      GB2 : Array[0..7480] of Word := [16#A1E8, 16#A1EC, 16#A1A7, 16#A1E3, 16#A1C0, 16#A1A4, 16#A1C1, 16#A8A4, 16#A8A2, 16#A8A8, 16#A8A6, 16#A8BA, 16#A8AC, 16#A8AA, 16#A8B0, 16#A8AE, 16#A1C2, 16#A8B4, 16#A8B2, 16#A8B9, 16#A8A1, 16#A8A5, 16#A8A7, 16#A8A9, 16#A8BD, 16#A8BE, 16#A8AD, 16#A8B1, 16#A8A3, 16#A8AB, 16#A8AF, 16#A8B3, 16#A8B5, 16#A8B6, 16#A8B7, 16#A8B8, 16#A8BB, 16#A8C0, 16#A1A6, 16#A1A5, 16#A6A1, 16#A6A2, 16#A6A3, 16#A6A4, 16#A6A5, 16#A6A6, 16#A6A7, 16#A6A8, 16#A6A9, 16#A6AA, 16#A6AB, 16#A6AC, 16#A6AD, 16#A6AE, 16#A6AF, 16#A6B0, 16#A6B1, 16#A6B2, 16#A6B3, 16#A6B4, 16#A6B5, 16#A6B6, 16#A6B7, 16#A6B8, 16#A6C1, 16#A6C2, 16#A6C3, 16#A6C4, 16#A6C5, 16#A6C6, 16#A6C7, 16#A6C8, 16#A6C9, 16#A6CA, 16#A6CB, 16#A6CC, 16#A6CD, 16#A6CE, 16#A6CF, 16#A6D0, 16#A6D1, 16#A6D2, 16#A6D3, 16#A6D4, 16#A6D5, 16#A6D6, 16#A6D7, 16#A6D8, 16#A7A7, 16#A7A1, 16#A7A2, 16#A7A3, 16#A7A4, 16#A7A5, 16#A7A6, 16#A7A8, 16#A7A9, 16#A7AA, 16#A7AB, 16#A7AC, 16#A7AD, 16#A7AE, 16#A7AF, 16#A7B0, 16#A7B1, 16#A7B2, 16#A7B3, 16#A7B4, 16#A7B5, 16#A7B6, 16#A7B7, 16#A7B8, 16#A7B9, 16#A7BA, 16#A7BB, 16#A7BC, 16#A7BD, 16#A7BE, 16#A7BF, 16#A7C0, 16#A7C1, 16#A7D1, 16#A7D2, 16#A7D3, 16#A7D4, 16#A7D5, 16#A7D6, 16#A7D8, 16#A7D9, 16#A7DA, 16#A7DB, 16#A7DC, 16#A7DD, 16#A7DE, 16#A7DF, 16#A7E0, 16#A7E1, 16#A7E2, 16#A7E3, 16#A7E4, 16#A7E5, 16#A7E6, 16#A7E7, 16#A7E8, 16#A7E9, 16#A7EA, 16#A7EB, 16#A7EC, 16#A7ED, 16#A7EE, 16#A7EF, 16#A7F0, 16#A7F1, 16#A7D7, 16#A1AA, 16#A1AC, 16#A1AE, 16#A1AF, 16#A1B0, 16#A1B1, 16#A1AD, 16#A1EB, 16#A1E4, 16#A1E5, 16#A1F9, 16#A1E6, 16#A1ED, 16#A2F1, 16#A2F2, 16#A2F3, 16#A2F4, 16#A2F5, 16#A2F6, 16#A2F7, 16#A2F8, 16#A2F9, 16#A2FA, 16#A2FB, 16#A2FC, 16#A2A1, 16#A2A2, 16#A2A3, 16#A2A4, 16#A2A5, 16#A2A6, 16#A2A7, 16#A2A8, 16#A2A9, 16#A2AA, 16#A1FB, 16#A1FC, 16#A1FA, 16#A1FD, 16#A1CA, 16#A1C7, 16#A1C6, 16#A1CC, 16#A1D8, 16#A1DE, 16#A1CF, 16#A1CE, 16#A1C4, 16#A1C5, 16#A1C9, 16#A1C8, 16#A1D2, 16#A1D3, 16#A1E0, 16#A1DF, 16#A1C3, 16#A1CB, 16#A1D7, 16#A1D6, 16#A1D5, 16#A1D9, 16#A1D4, 16#A1DC, 16#A1DD, 16#A1DA, 16#A1DB, 16#A1D1, 16#A1CD, 16#A1D0, 16#A2D9, 16#A2DA, 16#A2DB, 16#A2DC, 16#A2DD, 16#A2DE, 16#A2DF, 16#A2E0, 16#A2E1, 16#A2E2, 16#A2C5, 16#A2C6, 16#A2C7, 16#A2C8, 16#A2C9, 16#A2CA, 16#A2CB, 16#A2CC, 16#A2CD, 16#A2CE, 16#A2CF, 16#A2D0, 16#A2D1, 16#A2D2, 16#A2D3, 16#A2D4, 16#A2D5, 16#A2D6, 16#A2D7, 16#A2D8, 16#A2B1, 16#A2B2, 16#A2B3, 16#A2B4, 16#A2B5, 16#A2B6, 16#A2B7, 16#A2B8, 16#A2B9, 16#A2BA, 16#A2BB, 16#A2BC, 16#A2BD, 16#A2BE, 16#A2BF, 16#A2C0, 16#A2C1, 16#A2C2, 16#A2C3, 16#A2C4, 16#A9A4, 16#A9A5, 16#A9A6, 16#A9A7, 16#A9A8, 16#A9A9, 16#A9AA, 16#A9AB, 16#A9AC, 16#A9AD, 16#A9AE, 16#A9AF, 16#A9B0, 16#A9B1, 16#A9B2, 16#A9B3, 16#A9B4, 16#A9B5, 16#A9B6, 16#A9B7, 16#A9B8, 16#A9B9, 16#A9BA, 16#A9BB, 16#A9BC, 16#A9BD, 16#A9BE, 16#A9BF, 16#A9C0, 16#A9C1, 16#A9C2, 16#A9C3, 16#A9C4, 16#A9C5, 16#A9C6, 16#A9C7, 16#A9C8, 16#A9C9, 16#A9CA, 16#A9CB, 16#A9CC, 16#A9CD, 16#A9CE, 16#A9CF, 16#A9D0, 16#A9D1, 16#A9D2, 16#A9D3, 16#A9D4, 16#A9D5, 16#A9D6, 16#A9D7, 16#A9D8, 16#A9D9, 16#A9DA, 16#A9DB, 16#A9DC, 16#A9DD, 16#A9DE, 16#A9DF, 16#A9E0, 16#A9E1, 16#A9E2, 16#A9E3, 16#A9E4, 16#A9E5, 16#A9E6, 16#A9E7, 16#A9E8, 16#A9E9, 16#A9EA, 16#A9EB, 16#A9EC, 16#A9ED, 16#A9EE, 16#A9EF, 16#A1F6, 16#A1F5, 16#A1F8, 16#A1F7, 16#A1F4, 16#A1F3, 16#A1F0, 16#A1F2, 16#A1F1, 16#A1EF, 16#A1EE, 16#A1E2, 16#A1E1, 16#A1A1, 16#A1A2, 16#A1A3, 16#A1A8, 16#A1A9, 16#A1B4, 16#A1B5, 16#A1B6, 16#A1B7, 16#A1B8, 16#A1B9, 16#A1BA, 16#A1BB, 16#A1BE, 16#A1BF, 16#A1FE, 16#A1B2, 16#A1B3, 16#A1BC, 16#A1BD, 16#A4A1, 16#A4A2, 16#A4A3, 16#A4A4, 16#A4A5, 16#A4A6, 16#A4A7, 16#A4A8, 16#A4A9, 16#A4AA, 16#A4AB, 16#A4AC, 16#A4AD, 16#A4AE, 16#A4AF, 16#A4B0, 16#A4B1, 16#A4B2, 16#A4B3, 16#A4B4, 16#A4B5, 16#A4B6, 16#A4B7, 16#A4B8, 16#A4B9, 16#A4BA, 16#A4BB, 16#A4BC, 16#A4BD, 16#A4BE, 16#A4BF, 16#A4C0, 16#A4C1, 16#A4C2, 16#A4C3, 16#A4C4, 16#A4C5, 16#A4C6, 16#A4C7, 16#A4C8, 16#A4C9, 16#A4CA, 16#A4CB, 16#A4CC, 16#A4CD, 16#A4CE, 16#A4CF, 16#A4D0, 16#A4D1, 16#A4D2, 16#A4D3, 16#A4D4, 16#A4D5, 16#A4D6, 16#A4D7, 16#A4D8, 16#A4D9, 16#A4DA, 16#A4DB, 16#A4DC, 16#A4DD, 16#A4DE, 16#A4DF, 16#A4E0, 16#A4E1, 16#A4E2, 16#A4E3, 16#A4E4, 16#A4E5, 16#A4E6, 16#A4E7, 16#A4E8, 16#A4E9, 16#A4EA, 16#A4EB, 16#A4EC, 16#A4ED, 16#A4EE, 16#A4EF, 16#A4F0, 16#A4F1, 16#A4F2, 16#A4F3, 16#A5A1, 16#A5A2, 16#A5A3, 16#A5A4, 16#A5A5, 16#A5A6, 16#A5A7, 16#A5A8, 16#A5A9, 16#A5AA, 16#A5AB, 16#A5AC, 16#A5AD, 16#A5AE, 16#A5AF, 16#A5B0, 16#A5B1, 16#A5B2, 16#A5B3, 16#A5B4, 16#A5B5, 16#A5B6, 16#A5B7, 16#A5B8, 16#A5B9, 16#A5BA, 16#A5BB, 16#A5BC, 16#A5BD, 16#A5BE, 16#A5BF, 16#A5C0, 16#A5C1, 16#A5C2, 16#A5C3, 16#A5C4, 16#A5C5, 16#A5C6, 16#A5C7, 16#A5C8, 16#A5C9, 16#A5CA, 16#A5CB, 16#A5CC, 16#A5CD, 16#A5CE, 16#A5CF, 16#A5D0, 16#A5D1, 16#A5D2, 16#A5D3, 16#A5D4, 16#A5D5, 16#A5D6, 16#A5D7, 16#A5D8, 16#A5D9, 16#A5DA, 16#A5DB, 16#A5DC, 16#A5DD, 16#A5DE, 16#A5DF, 16#A5E0, 16#A5E1, 16#A5E2, 16#A5E3, 16#A5E4, 16#A5E5, 16#A5E6, 16#A5E7, 16#A5E8, 16#A5E9, 16#A5EA, 16#A5EB, 16#A5EC, 16#A5ED, 16#A5EE, 16#A5EF, 16#A5F0, 16#A5F1, 16#A5F2, 16#A5F3, 16#A5F4, 16#A5F5, 16#A5F6, 16#A8C5, 16#A8C6, 16#A8C7, 16#A8C8, 16#A8C9, 16#A8CA, 16#A8CB, 16#A8CC, 16#A8CD, 16#A8CE, 16#A8CF, 16#A8D0, 16#A8D1, 16#A8D2, 16#A8D3, 16#A8D4, 16#A8D5, 16#A8D6, 16#A8D7, 16#A8D8, 16#A8D9, 16#A8DA, 16#A8DB, 16#A8DC, 16#A8DD, 16#A8DE, 16#A8DF, 16#A8E0, 16#A8E1, 16#A8E2, 16#A8E3, 16#A8E4, 16#A8E5, 16#A8E6, 16#A8E7, 16#A8E8, 16#A8E9, 16#A2E5, 16#A2E6, 16#A2E7, 16#A2E8, 16#A2E9, 16#A2EA, 16#A2EB, 16#A2EC, 16#A2ED, 16#A2EE, 16#D2BB, 16#B6A1, 16#C6DF, 16#CDF2, 16#D5C9, 16#C8FD, 16#C9CF, 16#CFC2, 16#D8A2, 16#B2BB, 16#D3EB, 16#D8A4, 16#B3F3, 16#D7A8, 16#C7D2, 16#D8A7, 16#CAC0, 16#C7F0, 16#B1FB, 16#D2B5, 16#B4D4, 16#B6AB, 16#CBBF, 16#D8A9, 16#B6AA, 16#C1BD, 16#D1CF, 16#C9A5, 16#D8AD, 16#B8F6, 16#D1BE, 16#E3DC, 16#D6D0, 16#B7E1, 16#B4AE, 16#C1D9, 16#D8BC, 16#CDE8, 16#B5A4, 16#CEAA, 16#D6F7, 16#C0F6, 16#BED9, 16#D8AF, 16#C4CB, 16#BEC3, 16#D8B1, 16#C3B4, 16#D2E5, 16#D6AE, 16#CEDA, 16#D5A7, 16#BAF5, 16#B7A6, 16#C0D6, 16#C6B9, 16#C5D2, 16#C7C7, 16#B9D4, 16#B3CB, 16#D2D2, 16#D8BF, 16#BEC5, 16#C6F2, 16#D2B2, 16#CFB0, 16#CFE7, 16#CAE9, 16#D8C0, 16#C2F2, 16#C2D2, 16#C8E9, 16#C7AC, 16#C1CB, 16#D3E8, 16#D5F9, 16#CAC2, 16#B6FE, 16#D8A1, 16#D3DA, 16#BFF7, 16#D4C6, 16#BBA5, 16#D8C1, 16#CEE5, 16#BEAE, 16#D8A8, 16#D1C7, 16#D0A9, 16#D8BD, 16#D9EF, 16#CDF6, 16#BFBA, 16#BDBB, 16#BAA5, 16#D2E0, 16#B2FA, 16#BAE0, 16#C4B6, 16#CFED, 16#BEA9, 16#CDA4, 16#C1C1, 16#C7D7, 16#D9F1, 16#D9F4, 16#C8CB, 16#D8E9, 16#D2DA, 16#CAB2, 16#C8CA, 16#D8EC, 16#D8EA, 16#D8C6, 16#BDF6, 16#C6CD, 16#B3F0, 16#D8EB, 16#BDF1, 16#BDE9, 16#C8D4, 16#B4D3, 16#C2D8, 16#B2D6, 16#D7D0, 16#CACB, 16#CBFB, 16#D5CC, 16#B8B6, 16#CFC9, 16#D9DA, 16#D8F0, 16#C7AA, 16#D8EE, 16#B4FA, 16#C1EE, 16#D2D4, 16#D8ED, 16#D2C7, 16#D8EF, 16#C3C7, 16#D1F6, 16#D6D9, 16#D8F2, 16#D8F5, 16#BCFE, 16#BCDB, 16#C8CE, 16#B7DD, 16#B7C2, 16#C6F3, 16#D8F8, 16#D2C1, 16#CEE9, 16#BCBF, 16#B7FC, 16#B7A5, 16#D0DD, 16#D6DA, 16#D3C5, 16#BBEF, 16#BBE1, 16#D8F1, 16#C9A1, 16#CEB0, 16#B4AB, 16#D8F3, 16#C9CB, 16#D8F6, 16#C2D7, 16#D8F7, 16#CEB1, 16#D8F9, 16#B2AE, 16#B9C0, 16#D9A3, 16#B0E9, 16#C1E6, 16#C9EC, 16#CBC5, 16#CBC6, 16#D9A4, 16#B5E8, 16#B5AB, 16#CEBB, 16#B5CD, 16#D7A1, 16#D7F4, 16#D3D3, 16#CCE5, 16#BACE, 16#D9A2, 16#D9DC, 16#D3E0, 16#D8FD, 16#B7F0, 16#D7F7, 16#D8FE, 16#D8FA, 16#D9A1, 16#C4E3, 16#D3B6, 16#D8F4, 16#D9DD, 16#D8FB, 16#C5E5, 16#C0D0, 16#D1F0, 16#B0DB, 16#BCD1, 16#D9A6, 16#D9A5, 16#D9AC, 16#D9AE, 16#D9AB, 16#CAB9, 16#D9A9, 16#D6B6, 16#B3DE, 16#D9A8, 16#C0FD, 16#CACC, 16#D9AA, 16#D9A7, 16#D9B0, 16#B6B1, 16#B9A9, 16#D2C0, 16#CFC0, 16#C2C2, 16#BDC4, 16#D5EC, 16#B2E0, 16#C7C8, 16#BFEB, 16#D9AD, 16#D9AF, 16#CEEA, 16#BAEE, 16#C7D6, 16#B1E3, 16#B4D9, 16#B6ED, 16#D9B4, 16#BFA1, 16#D9DE, 16#C7CE, 16#C0FE, 16#D9B8, 16#CBD7, 16#B7FD, 16#D9B5, 16#D9B7, 16#B1A3, 16#D3E1, 16#D9B9, 16#D0C5, 16#D9B6, 16#D9B1, 16#D9B2, 16#C1A9, 16#D9B3, 16#BCF3, 16#D0DE, 16#B8A9, 16#BEE3, 16#D9BD, 16#D9BA, 16#B0B3, 16#D9C2, 16#D9C4, 16#B1B6, 16#D9BF, 16#B5B9, 16#BEF3, 16#CCC8, 16#BAF2, 16#D2D0, 16#D9C3, 16#BDE8, 16#B3AB, 16#D9C5, 16#BEEB, 16#D9C6, 16#D9BB, 16#C4DF, 16#D9BE, 16#D9C1, 16#D9C0, 16#D5AE, 16#D6B5, 16#C7E3, 16#D9C8, 16#BCD9, 16#D9CA, 16#D9BC, 16#D9CB, 16#C6AB, 16#D9C9, 16#D7F6, 16#CDA3, 16#BDA1, 16#D9CC, 16#C5BC, 16#CDB5, 16#D9CD, 16#D9C7, 16#B3A5, 16#BFFE, 16#B8B5, 16#C0FC, 16#B0F8, 16#B4F6, 16#D9CE, 16#D9CF, 16#B4A2, 16#D9D0, 16#B4DF, 16#B0C1, 16#D9D1, 16#C9B5, 16#CFF1, 16#D9D2, 16#C1C5, 16#D9D6, 16#C9AE, 16#D9D5, 16#D9D4, 16#D9D7, 16#CBDB, 16#BDA9, 16#C6A7, 16#D9D3, 16#D9D8, 16#D9D9, 16#C8E5, 16#C0DC, 16#B6F9, 16#D8A3, 16#D4CA, 16#D4AA, 16#D0D6, 16#B3E4, 16#D5D7, 16#CFC8, 16#B9E2, 16#BFCB, 16#C3E2, 16#B6D2, 16#CDC3, 16#D9EE, 16#D9F0, 16#B5B3, 16#B6B5, 16#BEA4, 16#C8EB, 16#C8AB, 16#B0CB, 16#B9AB, 16#C1F9, 16#D9E2, 16#C0BC, 16#B9B2, 16#B9D8, 16#D0CB, 16#B1F8, 16#C6E4, 16#BEDF, 16#B5E4, 16#D7C8, 16#D1F8, 16#BCE6, 16#CADE, 16#BCBD, 16#D9E6, 16#D8E7, 16#C4DA, 16#B8D4, 16#C8BD, 16#B2E1, 16#D4D9, 16#C3B0, 16#C3E1, 16#DAA2, 16#C8DF, 16#D0B4, 16#BEFC, 16#C5A9, 16#B9DA, 16#DAA3, 16#D4A9, 16#DAA4, 16#D9FB, 16#B6AC, 16#B7EB, 16#B1F9, 16#D9FC, 16#B3E5, 16#BEF6, 16#BFF6, 16#D2B1, 16#C0E4, 16#B6B3, 16#D9FE, 16#D9FD, 16#BEBB, 16#C6E0, 16#D7BC, 16#DAA1, 16#C1B9, 16#B5F2, 16#C1E8, 16#BCF5, 16#B4D5, 16#C1DD, 16#C4FD, 16#BCB8, 16#B7B2, 16#B7EF, 16#D9EC, 16#C6BE, 16#BFAD, 16#BBCB, 16#B5CA, 16#DBC9, 16#D0D7, 16#CDB9, 16#B0BC, 16#B3F6, 16#BBF7, 16#DBCA, 16#BAAF, 16#D4E4, 16#B5B6, 16#B5F3, 16#D8D6, 16#C8D0, 16#B7D6, 16#C7D0, 16#D8D7, 16#BFAF, 16#DBBB, 16#D8D8, 16#D0CC, 16#BBAE, 16#EBBE, 16#C1D0, 16#C1F5, 16#D4F2, 16#B8D5, 16#B4B4, 16#B3F5, 16#C9BE, 16#C5D0, 16#C5D9, 16#C0FB, 16#B1F0, 16#D8D9, 16#B9CE, 16#B5BD, 16#D8DA, 16#D6C6, 16#CBA2, 16#C8AF, 16#C9B2, 16#B4CC, 16#BFCC, 16#B9F4, 16#D8DB, 16#D8DC, 16#B6E7, 16#BCC1, 16#CCEA, 16#CFF7, 16#D8DD, 16#C7B0, 16#B9D0, 16#BDA3, 16#CCDE, 16#C6CA, 16#D8E0, 16#D8DE, 16#D8DF, 16#B0FE, 16#BEE7, 16#CAA3, 16#BCF4, 16#B8B1, 16#B8EE, 16#D8E2, 16#BDCB, 16#D8E4, 16#D8E3, 16#C5FC, 16#D8E5, 16#D8E6, 16#C1A6, 16#C8B0, 16#B0EC, 16#B9A6, 16#BCD3, 16#CEF1, 16#DBBD, 16#C1D3, 16#B6AF, 16#D6FA, 16#C5AC, 16#BDD9, 16#DBBE, 16#DBBF, 16#C0F8, 16#BEA2, 16#C0CD, 16#DBC0, 16#CAC6, 16#B2AA, 16#D3C2, 16#C3E3, 16#D1AB, 16#DBC2, 16#C0D5, 16#DBC3, 16#BFB1, 16#C4BC, 16#C7DA, 16#DBC4, 16#D9E8, 16#C9D7, 16#B9B4, 16#CEF0, 16#D4C8, 16#B0FC, 16#B4D2, 16#D0D9, 16#D9E9, 16#DECB, 16#D9EB, 16#D8B0, 16#BBAF, 16#B1B1, 16#B3D7, 16#D8CE, 16#D4D1, 16#BDB3, 16#BFEF, 16#CFBB, 16#D8D0, 16#B7CB, 16#D8D1, 16#C6A5, 16#C7F8, 16#D2BD, 16#D8D2, 16#C4E4, 16#CAAE, 16#C7A7, 16#D8A6, 16#C9FD, 16#CEE7, 16#BBDC, 16#B0EB, 16#BBAA, 16#D0AD, 16#B1B0, 16#D7E4, 16#D7BF, 16#B5A5, 16#C2F4, 16#C4CF, 16#B2A9, 16#B2B7, 16#B1E5, 16#DFB2, 16#D5BC, 16#BFA8, 16#C2AC, 16#D8D5, 16#C2B1, 16#D8D4, 16#CED4, 16#DAE0, 16#CEC0, 16#D8B4, 16#C3AE, 16#D3A1, 16#CEA3, 16#BCB4, 16#C8B4, 16#C2D1, 16#BEED, 16#D0B6, 16#DAE1, 16#C7E4, 16#B3A7, 16#B6F2, 16#CCFC, 16#C0FA, 16#C0F7, 16#D1B9, 16#D1E1, 16#D8C7, 16#B2DE, 16#C0E5, 16#BAF1, 16#D8C8, 16#D4AD, 16#CFE1, 16#D8C9, 16#D8CA, 16#CFC3, 16#B3F8, 16#BEC7, 16#D8CB, 16#DBCC, 16#C8A5, 16#CFD8, 16#C8FE, 16#B2CE, 16#D3D6, 16#B2E6, 16#BCB0, 16#D3D1, 16#CBAB, 16#B7B4, 16#B7A2, 16#CAE5, 16#C8A1, 16#CADC, 16#B1E4, 16#D0F0, 16#C5D1, 16#DBC5, 16#B5FE, 16#BFDA, 16#B9C5, 16#BEE4, 16#C1ED, 16#DFB6, 16#DFB5, 16#D6BB, 16#BDD0, 16#D5D9, 16#B0C8, 16#B6A3, 16#BFC9, 16#CCA8, 16#DFB3, 16#CAB7, 16#D3D2, 16#D8CF, 16#D2B6, 16#BAC5, 16#CBBE, 16#CCBE, 16#DFB7, 16#B5F0, 16#DFB4, 16#D3F5, 16#B3D4, 16#B8F7, 16#DFBA, 16#BACF, 16#BCAA, 16#B5F5, 16#CDAC, 16#C3FB, 16#BAF3, 16#C0F4, 16#CDC2, 16#CFF2, 16#DFB8, 16#CFC5, 16#C2C0, 16#DFB9, 16#C2F0, 16#BEFD, 16#C1DF, 16#CDCC, 16#D2F7, 16#B7CD, 16#DFC1, 16#DFC4, 16#B7F1, 16#B0C9, 16#B6D6, 16#B7D4, 16#BAAC, 16#CCFD, 16#BFD4, 16#CBB1, 16#C6F4, 16#D6A8, 16#DFC5, 16#CEE2, 16#B3B3, 16#CEFC, 16#B4B5, 16#CEC7, 16#BAF0, 16#CEE1, 16#D1BD, 16#DFC0, 16#B4F4, 16#B3CA, 16#B8E6, 16#DFBB, 16#C4C5, 16#DFBC, 16#DFBD, 16#DFBE, 16#C5BB, 16#DFBF, 16#DFC2, 16#D4B1, 16#DFC3, 16#C7BA, 16#CED8, 16#C4D8, 16#DFCA, 16#DFCF, 16#D6DC, 16#DFC9, 16#DFDA, 16#CEB6, 16#BAC7, 16#DFCE, 16#DFC8, 16#C5DE, 16#C9EB, 16#BAF4, 16#C3FC, 16#BED7, 16#DFC6, 16#DFCD, 16#C5D8, 16#D5A6, 16#BACD, 16#BECC, 16#D3BD, 16#B8C0, 16#D6E4, 16#DFC7, 16#B9BE, 16#BFA7, 16#C1FC, 16#DFCB, 16#DFCC, 16#DFD0, 16#DFDB, 16#DFE5, 16#DFD7, 16#DFD6, 16#D7C9, 16#DFE3, 16#DFE4, 16#E5EB, 16#D2A7, 16#DFD2, 16#BFA9, 16#D4DB, 16#BFC8, 16#DFD4, 16#CFCC, 16#DFDD, 16#D1CA, 16#DFDE, 16#B0A7, 16#C6B7, 16#DFD3, 16#BAE5, 16#B6DF, 16#CDDB, 16#B9FE, 16#D4D5, 16#DFDF, 16#CFEC, 16#B0A5, 16#DFE7, 16#DFD1, 16#D1C6, 16#DFD5, 16#DFD8, 16#DFD9, 16#DFDC, 16#BBA9, 16#DFE0, 16#DFE1, 16#DFE2, 16#DFE6, 16#DFE8, 16#D3B4, 16#B8E7, 16#C5B6, 16#DFEA, 16#C9DA, 16#C1A8, 16#C4C4, 16#BFDE, 16#CFF8, 16#D5DC, 16#DFEE, 16#B2B8, 16#BADF, 16#DFEC, 16#DBC1, 16#D1E4, 16#CBF4, 16#B4BD, 16#B0A6, 16#DFF1, 16#CCC6, 16#DFF2, 16#DFED, 16#DFE9, 16#DFEB, 16#DFEF, 16#DFF0, 16#BBBD, 16#DFF3, 16#DFF4, 16#BBA3, 16#CADB, 16#CEA8, 16#E0A7, 16#B3AA, 16#E0A6, 16#E0A1, 16#DFFE, 16#CDD9, 16#DFFC, 16#DFFA, 16#BFD0, 16#D7C4, 16#C9CC, 16#DFF8, 16#B0A1, 16#DFFD, 16#DFFB, 16#E0A2, 16#E0A8, 16#B7C8, 16#C6A1, 16#C9B6, 16#C0B2, 16#DFF5, 16#C5BE, 16#D8C4, 16#DFF9, 16#C4F6, 16#E0A3, 16#E0A4, 16#E0A5, 16#D0A5, 16#E0B4, 16#CCE4, 16#E0B1, 16#BFA6, 16#E0AF, 16#CEB9, 16#E0AB, 16#C9C6, 16#C0AE, 16#E0AE, 16#BAED, 16#BAB0, 16#E0A9, 16#DFF6, 16#E0B3, 16#E0B8, 16#B4AD, 16#E0B9, 16#CFB2, 16#BAC8, 16#E0B0, 16#D0FA, 16#E0AC, 16#D4FB, 16#DFF7, 16#C5E7, 16#E0AD, 16#D3F7, 16#E0B6, 16#E0B7, 16#E0C4, 16#D0E1, 16#E0BC, 16#E0C9, 16#E0CA, 16#E0BE, 16#E0AA, 16#C9A4, 16#E0C1, 16#E0B2, 16#CAC8, 16#E0C3, 16#E0B5, 16#CECB, 16#CBC3, 16#E0CD, 16#E0C6, 16#E0C2, 16#E0CB, 16#E0BA, 16#E0BF, 16#E0C0, 16#E0C5, 16#E0C7, 16#E0C8, 16#E0CC, 16#E0BB, 16#CBD4, 16#E0D5, 16#E0D6, 16#E0D2, 16#E0D0, 16#BCCE, 16#E0D1, 16#B8C2, 16#D8C5, 16#D0EA, 16#C2EF, 16#E0CF, 16#E0BD, 16#E0D4, 16#E0D3, 16#E0D7, 16#E0DC, 16#E0D8, 16#D6F6, 16#B3B0, 16#D7EC, 16#CBBB, 16#E0DA, 16#CEFB, 16#BAD9, 16#E0E1, 16#E0DD, 16#D2AD, 16#E0E2, 16#E0DB, 16#E0D9, 16#E0DF, 16#E0E0, 16#E0DE, 16#E0E4, 16#C6F7, 16#D8AC, 16#D4EB, 16#E0E6, 16#CAC9, 16#E0E5, 16#B8C1, 16#E0E7, 16#E0E8, 16#E0E9, 16#E0E3, 16#BABF, 16#CCE7, 16#E0EA, 16#CFF9, 16#E0EB, 16#C8C2, 16#BDC0, 16#C4D2, 16#E0EC, 16#E0ED, 16#C7F4, 16#CBC4, 16#E0EE, 16#BBD8, 16#D8B6, 16#D2F2, 16#E0EF, 16#CDC5, 16#B6DA, 16#E0F1, 16#D4B0, 16#C0A7, 16#B4D1, 16#CEA7, 16#E0F0, 16#E0F2, 16#B9CC, 16#B9FA, 16#CDBC, 16#E0F3, 16#C6D4, 16#E0F4, 16#D4B2, 16#C8A6, 16#E0F6, 16#E0F5, 16#E0F7, 16#CDC1, 16#CAA5, 16#D4DA, 16#DBD7, 16#DBD9, 16#DBD8, 16#B9E7, 16#DBDC, 16#DBDD, 16#B5D8, 16#DBDA, 16#DBDB, 16#B3A1, 16#DBDF, 16#BBF8, 16#D6B7, 16#DBE0, 16#BEF9, 16#B7BB, 16#DBD0, 16#CCAE, 16#BFB2, 16#BBB5, 16#D7F8, 16#BFD3, 16#BFE9, 16#BCE1, 16#CCB3, 16#DBDE, 16#B0D3, 16#CEEB, 16#B7D8, 16#D7B9, 16#C6C2, 16#C0A4, 16#CCB9, 16#DBE7, 16#DBE1, 16#C6BA, 16#DBE3, 16#DBE8, 16#C5F7, 16#DBEA, 16#DBE9, 16#BFC0, 16#DBE6, 16#DBE5, 16#B4B9, 16#C0AC, 16#C2A2, 16#DBE2, 16#DBE4, 16#D0CD, 16#DBED, 16#C0DD, 16#DBF2, 16#B6E2, 16#DBF3, 16#DBD2, 16#B9B8, 16#D4AB, 16#DBEC, 16#BFD1, 16#DBF0, 16#DBD1, 16#B5E6, 16#DBEB, 16#BFE5, 16#DBEE, 16#DBF1, 16#DBF9, 16#B9A1, 16#B0A3, 16#C2F1, 16#B3C7, 16#DBEF, 16#DBF8, 16#C6D2, 16#DBF4, 16#DBF5, 16#DBF7, 16#DBF6, 16#DBFE, 16#D3F2, 16#B2BA, 16#DBFD, 16#DCA4, 16#DBFB, 16#DBFA, 16#DBFC, 16#C5E0, 16#BBF9, 16#DCA3, 16#DCA5, 16#CCC3, 16#B6D1, 16#DDC0, 16#DCA1, 16#DCA2, 16#C7B5, 16#B6E9, 16#DCA7, 16#DCA6, 16#DCA9, 16#B1A4, 16#B5CC, 16#BFB0, 16#D1DF, 16#B6C2, 16#DCA8, 16#CBFA, 16#EBF3, 16#CBDC, 16#CBFE, 16#CCC1, 16#C8FB, 16#DCAA, 16#CCEE, 16#DCAB, 16#DBD3, 16#DCAF, 16#DCAC, 16#BEB3, 16#CAFB, 16#DCAD, 16#C9CA, 16#C4B9, 16#C7BD, 16#DCAE, 16#D4F6, 16#D0E6, 16#C4AB, 16#B6D5, 16#DBD4, 16#B1DA, 16#DBD5, 16#DBD6, 16#BABE, 16#C8C0, 16#CABF, 16#C8C9, 16#D7B3, 16#C9F9, 16#BFC7, 16#BAF8, 16#D2BC, 16#E2BA, 16#B4A6, 16#B1B8, 16#B8B4, 16#CFC4, 16#D9E7, 16#CFA6, 16#CDE2, 16#D9ED, 16#B6E0, 16#D2B9, 16#B9BB, 16#E2B9, 16#E2B7, 16#B4F3, 16#CCEC, 16#CCAB, 16#B7F2, 16#D8B2, 16#D1EB, 16#BABB, 16#CAA7, 16#CDB7, 16#D2C4, 16#BFE4, 16#BCD0, 16#B6E1, 16#DEC5, 16#DEC6, 16#DBBC, 16#D1D9, 16#C6E6, 16#C4CE, 16#B7EE, 16#B7DC, 16#BFFC, 16#D7E0, 16#C6F5, 16#B1BC, 16#DEC8, 16#BDB1, 16#CCD7, 16#DECA, 16#DEC9, 16#B5EC, 16#C9DD, 16#B0C2, 16#C5AE, 16#C5AB, 16#C4CC, 16#BCE9, 16#CBFD, 16#BAC3, 16#E5F9, 16#C8E7, 16#E5FA, 16#CDFD, 16#D7B1, 16#B8BE, 16#C2E8, 16#C8D1, 16#E5FB, 16#B6CA, 16#BCCB, 16#D1FD, 16#E6A1, 16#C3EE, 16#E6A4, 16#E5FE, 16#E6A5, 16#CDD7, 16#B7C1, 16#E5FC, 16#E5FD, 16#E6A3, 16#C4DD, 16#E6A8, 16#E6A7, 16#C3C3, 16#C6DE, 16#E6AA, 16#C4B7, 16#E6A2, 16#CABC, 16#BDE3, 16#B9C3, 16#E6A6, 16#D0D5, 16#CEAF, 16#E6A9, 16#E6B0, 16#D2A6, 16#BDAA, 16#E6AD, 16#E6AF, 16#C0D1, 16#D2CC, 16#BCA7, 16#E6B1, 16#D2F6, 16#D7CB, 16#CDFE, 16#CDDE, 16#C2A6, 16#E6AB, 16#E6AC, 16#BDBF, 16#E6AE, 16#E6B3, 16#E6B2, 16#E6B6, 16#E6B8, 16#C4EF, 16#C4C8, 16#BEEA, 16#C9EF, 16#E6B7, 16#B6F0, 16#C3E4, 16#D3E9, 16#E6B4, 16#E6B5, 16#C8A2, 16#E6BD, 16#E6B9, 16#C6C5, 16#CDF1, 16#E6BB, 16#E6BC, 16#BBE9, 16#E6BE, 16#E6BA, 16#C0B7, 16#D3A4, 16#E6BF, 16#C9F4, 16#E6C3, 16#E6C4, 16#D0F6, 16#C3BD, 16#C3C4, 16#E6C2, 16#E6C1, 16#E6C7, 16#CFB1, 16#EBF4, 16#E6CA, 16#E6C5, 16#BCDE, 16#C9A9, 16#BCB5, 16#CFD3, 16#E6C8, 16#E6C9, 16#E6CE, 16#E6D0, 16#E6D1, 16#E6CB, 16#B5D5, 16#E6CC, 16#E6CF, 16#C4DB, 16#E6C6, 16#E6CD, 16#E6D2, 16#E6D4, 16#E6D3, 16#E6D5, 16#D9F8, 16#E6D6, 16#E6D7, 16#D7D3, 16#E6DD, 16#E6DE, 16#BFD7, 16#D4D0, 16#D7D6, 16#B4E6, 16#CBEF, 16#E6DA, 16#D8C3, 16#D7CE, 16#D0A2, 16#C3CF, 16#E6DF, 16#BCBE, 16#B9C2, 16#E6DB, 16#D1A7, 16#BAA2, 16#C2CF, 16#D8AB, 16#CAEB, 16#E5EE, 16#E6DC, 16#B7F5, 16#C8E6, 16#C4F5, 16#E5B2, 16#C4FE, 16#CBFC, 16#E5B3, 16#D5AC, 16#D3EE, 16#CAD8, 16#B0B2, 16#CBCE, 16#CDEA, 16#BAEA, 16#E5B5, 16#E5B4, 16#D7DA, 16#B9D9, 16#D6E6, 16#B6A8, 16#CDF0, 16#D2CB, 16#B1A6, 16#CAB5, 16#B3E8, 16#C9F3, 16#BFCD, 16#D0FB, 16#CAD2, 16#E5B6, 16#BBC2, 16#CFDC, 16#B9AC, 16#D4D7, 16#BAA6, 16#D1E7, 16#CFFC, 16#BCD2, 16#E5B7, 16#C8DD, 16#BFED, 16#B1F6, 16#CBDE, 16#BCC5, 16#BCC4, 16#D2FA, 16#C3DC, 16#BFDC, 16#B8BB, 16#C3C2, 16#BAAE, 16#D4A2, 16#C7DE, 16#C4AF, 16#B2EC, 16#B9D1, 16#E5BB, 16#C1C8, 16#D5AF, 16#E5BC, 16#E5BE, 16#B4E7, 16#B6D4, 16#CBC2, 16#D1B0, 16#B5BC, 16#CAD9, 16#B7E2, 16#C9E4, 16#BDAB, 16#CEBE, 16#D7F0, 16#D0A1, 16#C9D9, 16#B6FB, 16#E6D8, 16#BCE2, 16#B3BE, 16#C9D0, 16#E6D9, 16#B3A2, 16#DECC, 16#D3C8, 16#DECD, 16#D2A2, 16#DECE, 16#BECD, 16#DECF, 16#CAAC, 16#D2FC, 16#B3DF, 16#E5EA, 16#C4E1, 16#BEA1, 16#CEB2, 16#C4F2, 16#BED6, 16#C6A8, 16#B2E3, 16#BED3, 16#C7FC, 16#CCEB, 16#BDEC, 16#CEDD, 16#CABA, 16#C6C1, 16#E5EC, 16#D0BC, 16#D5B9, 16#E5ED, 16#CAF4, 16#CDC0, 16#C2C5, 16#E5EF, 16#C2C4, 16#E5F0, 16#E5F8, 16#CDCD, 16#C9BD, 16#D2D9, 16#E1A8, 16#D3EC, 16#CBEA, 16#C6F1, 16#E1AC, 16#E1A7, 16#E1A9, 16#E1AA, 16#E1AF, 16#B2ED, 16#E1AB, 16#B8DA, 16#E1AD, 16#E1AE, 16#E1B0, 16#B5BA, 16#E1B1, 16#E1B3, 16#E1B8, 16#D1D2, 16#E1B6, 16#E1B5, 16#C1EB, 16#E1B7, 16#D4C0, 16#E1B2, 16#E1BA, 16#B0B6, 16#E1B4, 16#BFF9, 16#E1B9, 16#E1BB, 16#E1BE, 16#E1BC, 16#D6C5, 16#CFBF, 16#E1BD, 16#E1BF, 16#C2CD, 16#B6EB, 16#D3F8, 16#C7CD, 16#B7E5, 16#BEFE, 16#E1C0, 16#E1C1, 16#E1C7, 16#B3E7, 16#C6E9, 16#B4DE, 16#D1C2, 16#E1C8, 16#E1C6, 16#E1C5, 16#E1C3, 16#E1C2, 16#B1C0, 16#D5B8, 16#E1C4, 16#E1CB, 16#E1CC, 16#E1CA, 16#EFFA, 16#E1D3, 16#E1D2, 16#C7B6, 16#E1C9, 16#E1CE, 16#E1D0, 16#E1D4, 16#E1D1, 16#E1CD, 16#E1CF, 16#E1D5, 16#E1D6, 16#E1D7, 16#E1D8, 16#E1DA, 16#E1DB, 16#CEA1, 16#E7DD, 16#B4A8, 16#D6DD, 16#D1B2, 16#B3B2, 16#B9A4, 16#D7F3, 16#C7C9, 16#BEDE, 16#B9AE, 16#CED7, 16#B2EE, 16#DBCF, 16#BCBA, 16#D2D1, 16#CBC8, 16#B0CD, 16#CFEF, 16#D9E3, 16#BDED, 16#B1D2, 16#CAD0, 16#B2BC, 16#CBA7, 16#B7AB, 16#CAA6, 16#CFA3, 16#E0F8, 16#D5CA, 16#E0FB, 16#E0FA, 16#C5C1, 16#CCFB, 16#C1B1, 16#E0F9, 16#D6E3, 16#B2AF, 16#D6C4, 16#B5DB, 16#B4F8, 16#D6A1, 16#CFAF, 16#B0EF, 16#E0FC, 16#E1A1, 16#B3A3, 16#E0FD, 16#E0FE, 16#C3B1, 16#C3DD, 16#E1A2, 16#B7F9, 16#BBCF, 16#E1A3, 16#C4BB, 16#E1A4, 16#E1A5, 16#E1A6, 16#B4B1, 16#B8C9, 16#C6BD, 16#C4EA, 16#B2A2, 16#D0D2, 16#E7DB, 16#BBC3, 16#D3D7, 16#D3C4, 16#B9E3, 16#E2CF, 16#D7AF, 16#C7EC, 16#B1D3, 16#B4B2, 16#E2D1, 16#D0F2, 16#C2AE, 16#E2D0, 16#BFE2, 16#D3A6, 16#B5D7, 16#E2D2, 16#B5EA, 16#C3ED, 16#B8FD, 16#B8AE, 16#C5D3, 16#B7CF, 16#E2D4, 16#E2D3, 16#B6C8, 16#D7F9, 16#CDA5, 16#E2D8, 16#E2D6, 16#CAFC, 16#BFB5, 16#D3B9, 16#E2D5, 16#E2D7, 16#C1AE, 16#C0C8, 16#E2DB, 16#E2DA, 16#C0AA, 16#C1CE, 16#E2DC, 16#E2DD, 16#E2DE, 16#DBC8, 16#D1D3, 16#CDA2, 16#BDA8, 16#DEC3, 16#D8A5, 16#BFAA, 16#DBCD, 16#D2EC, 16#C6FA, 16#C5AA, 16#DEC4, 16#B1D7, 16#DFAE, 16#CABD, 16#DFB1, 16#B9AD, 16#D2FD, 16#B8A5, 16#BAEB, 16#B3DA, 16#B5DC, 16#D5C5, 16#C3D6, 16#CFD2, 16#BBA1, 16#E5F3, 16#E5F2, 16#E5F4, 16#CDE4, 16#C8F5, 16#B5AF, 16#C7BF, 16#E5F6, 16#ECB0, 16#E5E6, 16#B9E9, 16#B5B1, 16#C2BC, 16#E5E8, 16#E5E7, 16#E5E9, 16#D2CD, 16#E1EA, 16#D0CE, 16#CDAE, 16#D1E5, 16#B2CA, 16#B1EB, 16#B1F2, 16#C5ED, 16#D5C3, 16#D3B0, 16#E1DC, 16#E1DD, 16#D2DB, 16#B3B9, 16#B1CB, 16#CDF9, 16#D5F7, 16#E1DE, 16#BEB6, 16#B4FD, 16#E1DF, 16#BADC, 16#E1E0, 16#BBB2, 16#C2C9, 16#E1E1, 16#D0EC, 16#CDBD, 16#E1E2, 16#B5C3, 16#C5C7, 16#E1E3, 16#E1E4, 16#D3F9, 16#E1E5, 16#D1AD, 16#E1E6, 16#CEA2, 16#E1E7, 16#B5C2, 16#E1E8, 16#BBD5, 16#D0C4, 16#E2E0, 16#B1D8, 16#D2E4, 16#E2E1, 16#BCC9, 16#C8CC, 16#E2E3, 16#ECFE, 16#ECFD, 16#DFAF, 16#E2E2, 16#D6BE, 16#CDFC, 16#C3A6, 16#E3C3, 16#D6D2, 16#E2E7, 16#E2E8, 16#D3C7, 16#E2EC, 16#BFEC, 16#E2ED, 16#E2E5, 16#B3C0, 16#C4EE, 16#E2EE, 16#D0C3, 16#BAF6, 16#E2E9, 16#B7DE, 16#BBB3, 16#CCAC, 16#CBCB, 16#E2E4, 16#E2E6, 16#E2EA, 16#E2EB, 16#E2F7, 16#E2F4, 16#D4F5, 16#E2F3, 16#C5AD, 16#D5FA, 16#C5C2, 16#B2C0, 16#E2EF, 16#E2F2, 16#C1AF, 16#CBBC, 16#B5A1, 16#E2F9, 16#BCB1, 16#E2F1, 16#D0D4, 16#D4B9, 16#E2F5, 16#B9D6, 16#E2F6, 16#C7D3, 16#E2F0, 16#D7DC, 16#EDA1, 16#E2F8, 16#EDA5, 16#E2FE, 16#CAD1, 16#C1B5, 16#BBD0, 16#BFD6, 16#BAE3, 16#CBA1, 16#EDA6, 16#EDA3, 16#EDA2, 16#BBD6, 16#EDA7, 16#D0F4, 16#EDA4, 16#BADE, 16#B6F7, 16#E3A1, 16#B6B2, 16#CCF1, 16#B9A7, 16#CFA2, 16#C7A1, 16#BFD2, 16#B6F1, 16#E2FA, 16#E2FB, 16#E2FD, 16#E2FC, 16#C4D5, 16#E3A2, 16#D3C1, 16#E3A7, 16#C7C4, 16#CFA4, 16#E3A9, 16#BAB7, 16#E3A8, 16#BBDA, 16#E3A3, 16#E3A4, 16#E3AA, 16#E3A6, 16#CEF2, 16#D3C6, 16#BBBC, 16#D4C3, 16#C4FA, 16#EDA8, 16#D0FC, 16#E3A5, 16#C3F5, 16#E3AD, 16#B1AF, 16#E3B2, 16#BCC2, 16#E3AC, 16#B5BF, 16#C7E9, 16#E3B0, 16#BEAA, 16#CDEF, 16#BBF3, 16#CCE8, 16#E3AF, 16#E3B1, 16#CFA7, 16#E3AE, 16#CEA9, 16#BBDD, 16#B5EB, 16#BEE5, 16#B2D2, 16#B3CD, 16#B1B9, 16#E3AB, 16#B2D1, 16#B5AC, 16#B9DF, 16#B6E8, 16#CFEB, 16#E3B7, 16#BBCC, 16#C8C7, 16#D0CA, 16#E3B8, 16#B3EE, 16#EDA9, 16#D3FA, 16#D3E4, 16#EDAA, 16#E3B9, 16#D2E2, 16#E3B5, 16#D3DE, 16#B8D0, 16#E3B3, 16#E3B6, 16#B7DF, 16#E3B4, 16#C0A2, 16#E3BA, 16#D4B8, 16#B4C8, 16#E3BB, 16#BBC5, 16#C9F7, 16#C9E5, 16#C4BD, 16#EDAB, 16#C2FD, 16#BBDB, 16#BFAE, 16#CEBF, 16#E3BC, 16#BFB6, 16#B1EF, 16#D4F7, 16#E3BE, 16#EDAD, 16#E3BF, 16#BAA9, 16#EDAC, 16#E3BD, 16#E3C0, 16#BAB6, 16#B6AE, 16#D0B8, 16#B0C3, 16#EDAE, 16#EDAF, 16#C0C1, 16#E3C1, 16#C5B3, 16#E3C2, 16#DCB2, 16#EDB0, 16#B8EA, 16#CEEC, 16#EAA7, 16#D0E7, 16#CAF9, 16#C8D6, 16#CFB7, 16#B3C9, 16#CED2, 16#BDE4, 16#E3DE, 16#BBF2, 16#EAA8, 16#D5BD, 16#C6DD, 16#EAA9, 16#EAAA, 16#EAAC, 16#EAAB, 16#EAAE, 16#EAAD, 16#BDD8, 16#EAAF, 16#C2BE, 16#B4C1, 16#B4F7, 16#BBA7, 16#ECE6, 16#ECE5, 16#B7BF, 16#CBF9, 16#B1E2, 16#ECE7, 16#C9C8, 16#ECE8, 16#ECE9, 16#CAD6, 16#DED0, 16#B2C5, 16#D4FA, 16#C6CB, 16#B0C7, 16#B4F2, 16#C8D3, 16#CDD0, 16#BFB8, 16#BFDB, 16#C7A4, 16#D6B4, 16#C0A9, 16#DED1, 16#C9A8, 16#D1EF, 16#C5A4, 16#B0E7, 16#B3B6, 16#C8C5, 16#B0E2, 16#B7F6, 16#C5FA, 16#B6F3, 16#D5D2, 16#B3D0, 16#BCBC, 16#B3AD, 16#BEF1, 16#B0D1, 16#D2D6, 16#CAE3, 16#D7A5, 16#CDB6, 16#B6B6, 16#BFB9, 16#D5DB, 16#B8A7, 16#C5D7, 16#DED2, 16#BFD9, 16#C2D5, 16#C7C0, 16#BBA4, 16#B1A8, 16#C5EA, 16#C5FB, 16#CCA7, 16#B1A7, 16#B5D6, 16#C4A8, 16#DED3, 16#D1BA, 16#B3E9, 16#C3F2, 16#B7F7, 16#D6F4, 16#B5A3, 16#B2F0, 16#C4B4, 16#C4E9, 16#C0AD, 16#DED4, 16#B0E8, 16#C5C4, 16#C1E0, 16#B9D5, 16#BEDC, 16#CDD8, 16#B0CE, 16#CDCF, 16#DED6, 16#BED0, 16#D7BE, 16#DED5, 16#D5D0, 16#B0DD, 16#C4E2, 16#C2A3, 16#BCF0, 16#D3B5, 16#C0B9, 16#C5A1, 16#B2A6, 16#D4F1, 16#C0A8, 16#CAC3, 16#DED7, 16#D5FC, 16#B9B0, 16#C8AD, 16#CBA9, 16#DED9, 16#BFBD, 16#C6B4, 16#D7A7, 16#CAB0, 16#C4C3, 16#B3D6, 16#B9D2, 16#D6B8, 16#EAFC, 16#B0B4, 16#BFE6, 16#CCF4, 16#CDDA, 16#D6BF, 16#C2CE, 16#CECE, 16#CCA2, 16#D0AE, 16#C4D3, 16#B5B2, 16#DED8, 16#D5F5, 16#BCB7, 16#BBD3, 16#B0A4, 16#C5B2, 16#B4EC, 16#D5F1, 16#EAFD, 16#DEDA, 16#CDA6, 16#CDEC, 16#CEE6, 16#DEDC, 16#CDB1, 16#C0A6, 16#D7BD, 16#DEDB, 16#B0C6, 16#BAB4, 16#C9D3, 16#C4F3, 16#BEE8, 16#B2B6, 16#C0CC, 16#CBF0, 16#BCF1, 16#BBBB, 16#B5B7, 16#C5F5, 16#DEE6, 16#DEE3, 16#BEDD, 16#DEDF, 16#B4B7, 16#BDDD, 16#DEE0, 16#C4ED, 16#CFC6, 16#B5E0, 16#B6DE, 16#CADA, 16#B5F4, 16#DEE5, 16#D5C6, 16#DEE1, 16#CCCD, 16#C6FE, 16#C5C5, 16#D2B4, 16#BEF2, 16#C2D3, 16#CCBD, 16#B3B8, 16#BDD3, 16#BFD8, 16#CDC6, 16#D1DA, 16#B4EB, 16#DEE4, 16#DEDD, 16#DEE7, 16#EAFE, 16#C2B0, 16#DEE2, 16#D6C0, 16#B5A7, 16#B2F4, 16#DEE8, 16#DEF2, 16#DEED, 16#DEF1, 16#C8E0, 16#D7E1, 16#DEEF, 16#C3E8, 16#CCE1, 16#B2E5, 16#D2BE, 16#DEEE, 16#DEEB, 16#CED5, 16#B4A7, 16#BFAB, 16#BEBE, 16#BDD2, 16#DEE9, 16#D4AE, 16#DEDE, 16#DEEA, 16#C0BF, 16#DEEC, 16#B2F3, 16#B8E9, 16#C2A7, 16#BDC1, 16#DEF5, 16#DEF8, 16#B2AB, 16#B4A4, 16#B4EA, 16#C9A6, 16#DEF6, 16#CBD1, 16#B8E3, 16#DEF7, 16#DEFA, 16#DEF9, 16#CCC2, 16#B0E1, 16#B4EE, 16#E5BA, 16#D0AF, 16#B2EB, 16#EBA1, 16#DEF4, 16#C9E3, 16#DEF3, 16#B0DA, 16#D2A1, 16#B1F7, 16#CCAF, 16#DEF0, 16#CBA4, 16#D5AA, 16#DEFB, 16#B4DD, 16#C4A6, 16#DEFD, 16#C3FE, 16#C4A1, 16#DFA1, 16#C1CC, 16#DEFC, 16#BEEF, 16#C6B2, 16#B3C5, 16#C8F6, 16#CBBA, 16#DEFE, 16#DFA4, 16#D7B2, 16#B3B7, 16#C1C3, 16#C7CB, 16#B2A5, 16#B4E9, 16#D7AB, 16#C4EC, 16#DFA2, 16#DFA3, 16#DFA5, 16#BAB3, 16#DFA6, 16#C0DE, 16#C9C3, 16#B2D9, 16#C7E6, 16#DFA7, 16#C7DC, 16#DFA8, 16#EBA2, 16#CBD3, 16#DFAA, 16#DFA9, 16#B2C1, 16#C5CA, 16#DFAB, 16#D4DC, 16#C8C1, 16#DFAC, 16#BEF0, 16#DFAD, 16#D6A7, 16#EAB7, 16#EBB6, 16#CAD5, 16#D8FC, 16#B8C4, 16#B9A5, 16#B7C5, 16#D5FE, 16#B9CA, 16#D0A7, 16#F4CD, 16#B5D0, 16#C3F4, 16#BEC8, 16#EBB7, 16#B0BD, 16#BDCC, 16#C1B2, 16#B1D6, 16#B3A8, 16#B8D2, 16#C9A2, 16#B6D8, 16#EBB8, 16#BEB4, 16#CAFD, 16#C7C3, 16#D5FB, 16#B7F3, 16#CEC4, 16#D5AB, 16#B1F3, 16#ECB3, 16#B0DF, 16#ECB5, 16#B6B7, 16#C1CF, 16#F5FA, 16#D0B1, 16#D5E5, 16#CED3, 16#BDEF, 16#B3E2, 16#B8AB, 16#D5B6, 16#EDBD, 16#B6CF, 16#CBB9, 16#D0C2, 16#B7BD, 16#ECB6, 16#CAA9, 16#C5D4, 16#ECB9, 16#ECB8, 16#C2C3, 16#ECB7, 16#D0FD, 16#ECBA, 16#ECBB, 16#D7E5, 16#ECBC, 16#ECBD, 16#C6EC, 16#CEDE, 16#BCC8, 16#C8D5, 16#B5A9, 16#BEC9, 16#D6BC, 16#D4E7, 16#D1AE, 16#D0F1, 16#EAB8, 16#EAB9, 16#EABA, 16#BAB5, 16#CAB1, 16#BFF5, 16#CDFA, 16#EAC0, 16#B0BA, 16#EABE, 16#C0A5, 16#EABB, 16#B2FD, 16#C3F7, 16#BBE8, 16#D2D7, 16#CEF4, 16#EABF, 16#EABC, 16#EAC3, 16#D0C7, 16#D3B3, 16#B4BA, 16#C3C1, 16#D7F2, 16#D5D1, 16#CAC7, 16#EAC5, 16#EAC4, 16#EAC7, 16#EAC6, 16#D6E7, 16#CFD4, 16#EACB, 16#BBCE, 16#BDFA, 16#C9CE, 16#EACC, 16#C9B9, 16#CFFE, 16#EACA, 16#D4CE, 16#EACD, 16#EACF, 16#CDED, 16#EAC9, 16#EACE, 16#CEEE, 16#BBDE, 16#B3BF, 16#C6D5, 16#BEB0, 16#CEFA, 16#C7E7, 16#BEA7, 16#EAD0, 16#D6C7, 16#C1C0, 16#D4DD, 16#EAD1, 16#CFBE, 16#EAD2, 16#CAEE, 16#C5AF, 16#B0B5, 16#EAD4, 16#EAD3, 16#F4DF, 16#C4BA, 16#B1A9, 16#E5DF, 16#EAD5, 16#CAEF, 16#EAD6, 16#EAD7, 16#C6D8, 16#EAD8, 16#EAD9, 16#D4BB, 16#C7FA, 16#D2B7, 16#B8FC, 16#EAC2, 16#B2DC, 16#C2FC, 16#D4F8, 16#CCE6, 16#D7EE, 16#D4C2, 16#D3D0, 16#EBC3, 16#C5F3, 16#B7FE, 16#EBD4, 16#CBB7, 16#EBDE, 16#C0CA, 16#CDFB, 16#B3AF, 16#C6DA, 16#EBFC, 16#C4BE, 16#CEB4, 16#C4A9, 16#B1BE, 16#D4FD, 16#CAF5, 16#D6EC, 16#C6D3, 16#B6E4, 16#BBFA, 16#D0E0, 16#C9B1, 16#D4D3, 16#C8A8, 16#B8CB, 16#E8BE, 16#C9BC, 16#E8BB, 16#C0EE, 16#D0D3, 16#B2C4, 16#B4E5, 16#E8BC, 16#D5C8, 16#B6C5, 16#E8BD, 16#CAF8, 16#B8DC, 16#CCF5, 16#C0B4, 16#D1EE, 16#E8BF, 16#E8C2, 16#BABC, 16#B1AD, 16#BDDC, 16#EABD, 16#E8C3, 16#E8C6, 16#E8CB, 16#E8CC, 16#CBC9, 16#B0E5, 16#BCAB, 16#B9B9, 16#E8C1, 16#CDF7, 16#E8CA, 16#CEF6, 16#D5ED, 16#C1D6, 16#E8C4, 16#C3B6, 16#B9FB, 16#D6A6, 16#E8C8, 16#CAE0, 16#D4E6, 16#E8C0, 16#E8C5, 16#E8C7, 16#C7B9, 16#B7E3, 16#E8C9, 16#BFDD, 16#E8D2, 16#E8D7, 16#E8D5, 16#BCDC, 16#BCCF, 16#E8DB, 16#E8DE, 16#E8DA, 16#B1FA, 16#B0D8, 16#C4B3, 16#B8CC, 16#C6E2, 16#C8BE, 16#C8E1, 16#E8CF, 16#E8D4, 16#E8D6, 16#B9F1, 16#E8D8, 16#D7F5, 16#C4FB, 16#E8DC, 16#B2E9, 16#E8D1, 16#BCED, 16#BFC2, 16#E8CD, 16#D6F9, 16#C1F8, 16#B2F1, 16#E8DF, 16#CAC1, 16#E8D9, 16#D5A4, 16#B1EA, 16#D5BB, 16#E8CE, 16#E8D0, 16#B6B0, 16#E8D3, 16#E8DD, 16#C0B8, 16#CAF7, 16#CBA8, 16#C6DC, 16#C0F5, 16#E8E9, 16#D0A3, 16#E8F2, 16#D6EA, 16#E8E0, 16#E8E1, 16#D1F9, 16#BACB, 16#B8F9, 16#B8F1, 16#D4D4, 16#E8EF, 16#E8EE, 16#E8EC, 16#B9F0, 16#CCD2, 16#E8E6, 16#CEA6, 16#BFF2, 16#B0B8, 16#E8F1, 16#E8F0, 16#D7C0, 16#E8E4, 16#CDA9, 16#C9A3, 16#BBB8, 16#BDDB, 16#E8EA, 16#E8E2, 16#E8E3, 16#E8E5, 16#B5B5, 16#E8E7, 16#C7C5, 16#E8EB, 16#E8ED, 16#BDB0, 16#D7AE, 16#E8F8, 16#E8F5, 16#CDB0, 16#E8F6, 16#C1BA, 16#E8E8, 16#C3B7, 16#B0F0, 16#E8F4, 16#E8F7, 16#B9A3, 16#C9D2, 16#C3CE, 16#CEE0, 16#C0E6, 16#CBF3, 16#CCDD, 16#D0B5, 16#CAE1, 16#E8F3, 16#BCEC, 16#E8F9, 16#C3DE, 16#C6E5, 16#B9F7, 16#B0F4, 16#D7D8, 16#BCAC, 16#C5EF, 16#CCC4, 16#E9A6, 16#C9AD, 16#E9A2, 16#C0E2, 16#BFC3, 16#E8FE, 16#B9D7, 16#E8FB, 16#E9A4, 16#D2CE, 16#E9A3, 16#D6B2, 16#D7B5, 16#E9A7, 16#BDB7, 16#E8FC, 16#E8FD, 16#E9A1, 16#CDD6, 16#D2AC, 16#E9B2, 16#E9A9, 16#B4AA, 16#B4BB, 16#E9AB, 16#D0A8, 16#E9A5, 16#B3FE, 16#E9AC, 16#C0E3, 16#E9AA, 16#E9B9, 16#E9B8, 16#E9AE, 16#E8FA, 16#E9A8, 16#BFAC, 16#E9B1, 16#E9BA, 16#C2A5, 16#E9AF, 16#B8C5, 16#E9AD, 16#D3DC, 16#E9B4, 16#E9B5, 16#E9B7, 16#E9C7, 16#C0C6, 16#E9C5, 16#E9B0, 16#E9BB, 16#B0F1, 16#E9BC, 16#D5A5, 16#E9BE, 16#E9BF, 16#E9C1, 16#C1F1, 16#C8B6, 16#E9BD, 16#E9C2, 16#E9C3, 16#E9B3, 16#E9B6, 16#BBB1, 16#E9C0, 16#BCF7, 16#E9C4, 16#E9C6, 16#E9CA, 16#E9CE, 16#B2DB, 16#E9C8, 16#B7AE, 16#E9CB, 16#E9CC, 16#D5C1, 16#C4A3, 16#E9D8, 16#BAE1, 16#E9C9, 16#D3A3, 16#E9D4, 16#E9D7, 16#E9D0, 16#E9CF, 16#C7C1, 16#E9D2, 16#E9D9, 16#B3C8, 16#E9D3, 16#CFF0, 16#E9CD, 16#B3F7, 16#E9D6, 16#E9DA, 16#CCB4, 16#CFAD, 16#E9D5, 16#E9DC, 16#E9DB, 16#E9DE, 16#E9D1, 16#E9DD, 16#E9DF, 16#C3CA, 16#C7B7, 16#B4CE, 16#BBB6, 16#D0C0, 16#ECA3, 16#C5B7, 16#D3FB, 16#ECA4, 16#ECA5, 16#C6DB, 16#BFEE, 16#ECA6, 16#ECA7, 16#D0AA, 16#C7B8, 16#B8E8, 16#ECA8, 16#D6B9, 16#D5FD, 16#B4CB, 16#B2BD, 16#CEE4, 16#C6E7, 16#CDE1, 16#B4F5, 16#CBC0, 16#BCDF, 16#E9E2, 16#E9E3, 16#D1EA, 16#E9E5, 16#B4F9, 16#E9E4, 16#D1B3, 16#CAE2, 16#B2D0, 16#E9E8, 16#E9E6, 16#E9E7, 16#D6B3, 16#E9E9, 16#E9EA, 16#E9EB, 16#E9EC, 16#ECAF, 16#C5B9, 16#B6CE, 16#D2F3, 16#B5EE, 16#BBD9, 16#ECB1, 16#D2E3, 16#CEE3, 16#C4B8, 16#C3BF, 16#B6BE, 16#D8B9, 16#B1C8, 16#B1CF, 16#B1D1, 16#C5FE, 16#B1D0, 16#C3AB, 16#D5B1, 16#EBA4, 16#BAC1, 16#CCBA, 16#EBA5, 16#EBA7, 16#EBA8, 16#EBA6, 16#EBA9, 16#EBAB, 16#EBAA, 16#EBAC, 16#CACF, 16#D8B5, 16#C3F1, 16#C3A5, 16#C6F8, 16#EBAD, 16#C4CA, 16#EBAE, 16#EBAF, 16#EBB0, 16#B7D5, 16#B7FA, 16#EBB1, 16#C7E2, 16#EBB3, 16#BAA4, 16#D1F5, 16#B0B1, 16#EBB2, 16#EBB4, 16#B5AA, 16#C2C8, 16#C7E8, 16#EBB5, 16#CBAE, 16#E3DF, 16#D3C0, 16#D9DB, 16#CDA1, 16#D6AD, 16#C7F3, 16#D9E0, 16#BBE3, 16#BABA, 16#E3E2, 16#CFAB, 16#E3E0, 16#C9C7, 16#BAB9, 16#D1B4, 16#E3E1, 16#C8EA, 16#B9AF, 16#BDAD, 16#B3D8, 16#CEDB, 16#CCC0, 16#E3E8, 16#E3E9, 16#CDF4, 16#CCAD, 16#BCB3, 16#E3EA, 16#E3EB, 16#D0DA, 16#C6FB, 16#B7DA, 16#C7DF, 16#D2CA, 16#CED6, 16#E3E4, 16#E3EC, 16#C9F2, 16#B3C1, 16#E3E7, 16#C6E3, 16#E3E5, 16#EDB3, 16#E3E6, 16#C9B3, 16#C5E6, 16#B9B5, 16#C3BB, 16#E3E3, 16#C5BD, 16#C1A4, 16#C2D9, 16#B2D7, 16#E3ED, 16#BBA6, 16#C4AD, 16#E3F0, 16#BEDA, 16#E3FB, 16#E3F5, 16#BAD3, 16#B7D0, 16#D3CD, 16#D6CE, 16#D5D3, 16#B9C1, 16#D5B4, 16#D1D8, 16#D0B9, 16#C7F6, 16#C8AA, 16#B2B4, 16#C3DA, 16#E3EE, 16#E3FC, 16#E3EF, 16#B7A8, 16#E3F7, 16#E3F4, 16#B7BA, 16#C5A2, 16#E3F6, 16#C5DD, 16#B2A8, 16#C6FC, 16#C4E0, 16#D7A2, 16#C0E1, 16#E3F9, 16#E3FA, 16#E3FD, 16#CCA9, 16#E3F3, 16#D3BE, 16#B1C3, 16#EDB4, 16#E3F1, 16#E3F2, 16#E3F8, 16#D0BA, 16#C6C3, 16#D4F3, 16#E3FE, 16#BDE0, 16#E4A7, 16#E4A6, 16#D1F3, 16#E4A3, 16#E4A9, 16#C8F7, 16#CFB4, 16#E4A8, 16#E4AE, 16#C2E5, 16#B6B4, 16#BDF2, 16#E4A2, 16#BAE9, 16#E4AA, 16#E4AC, 16#B6FD, 16#D6DE, 16#E4B2, 16#E4AD, 16#E4A1, 16#BBEE, 16#CDDD, 16#C7A2, 16#C5C9, 16#C1F7, 16#E4A4, 16#C7B3, 16#BDAC, 16#BDBD, 16#E4A5, 16#D7C7, 16#B2E2, 16#E4AB, 16#BCC3, 16#E4AF, 16#BBEB, 16#E4B0, 16#C5A8, 16#E4B1, 16#D5E3, 16#BFA3, 16#E4BA, 16#E4B7, 16#E4BB, 16#E4BD, 16#C6D6, 16#BAC6, 16#C0CB, 16#B8A1, 16#E4B4, 16#D4A1, 16#BAA3, 16#BDFE, 16#E4BC, 16#CDBF, 16#C4F9, 16#CFFB, 16#C9E6, 16#D3BF, 16#CFD1, 16#E4B3, 16#E4B8, 16#E4B9, 16#CCE9, 16#CCCE, 16#C0D4, 16#E4B5, 16#C1B0, 16#E4B6, 16#CED0, 16#BBC1, 16#B5D3, 16#C8F3, 16#BDA7, 16#D5C7, 16#C9AC, 16#B8A2, 16#E4CA, 16#E4CC, 16#D1C4, 16#D2BA, 16#BAAD, 16#BAD4, 16#E4C3, 16#B5ED, 16#D7CD, 16#E4C0, 16#CFFD, 16#E4BF, 16#C1DC, 16#CCCA, 16#CAE7, 16#C4D7, 16#CCD4, 16#E4C8, 16#E4C7, 16#E4C1, 16#E4C4, 16#B5AD, 16#D3D9, 16#E4C6, 16#D2F9, 16#B4E3, 16#BBB4, 16#C9EE, 16#B4BE, 16#BBEC, 16#D1CD, 16#CCED, 16#EDB5, 16#C7E5, 16#D4A8, 16#E4CB, 16#D7D5, 16#E4C2, 16#BDA5, 16#E4C5, 16#D3E6, 16#E4C9, 16#C9F8, 16#E4BE, 16#D3E5, 16#C7FE, 16#B6C9, 16#D4FC, 16#B2B3, 16#E4D7, 16#CEC2, 16#E4CD, 16#CEBC, 16#B8DB, 16#E4D6, 16#BFCA, 16#D3CE, 16#C3EC, 16#C5C8, 16#E4D8, 16#CDC4, 16#E4CF, 16#E4D4, 16#E4D5, 16#BAFE, 16#CFE6, 16#D5BF, 16#E4D2, 16#E4D0, 16#E4CE, 16#CDE5, 16#CAAA, 16#C0A3, 16#BDA6, 16#E4D3, 16#B8C8, 16#E4E7, 16#D4B4, 16#E4DB, 16#C1EF, 16#E4E9, 16#D2E7, 16#E4DF, 16#E4E0, 16#CFAA, 16#CBDD, 16#E4DA, 16#E4D1, 16#E4E5, 16#C8DC, 16#E4E3, 16#C4E7, 16#E4E2, 16#E4E1, 16#B3FC, 16#E4E8, 16#B5E1, 16#D7CC, 16#E4E6, 16#BBAC, 16#D7D2, 16#CCCF, 16#EBF8, 16#E4E4, 16#B9F6, 16#D6CD, 16#E4D9, 16#E4DC, 16#C2FA, 16#E4DE, 16#C2CB, 16#C0C4, 16#C2D0, 16#B1F5, 16#CCB2, 16#B5CE, 16#E4EF, 16#C6AF, 16#C6E1, 16#E4F5, 16#C2A9, 16#C0EC, 16#D1DD, 16#E4EE, 16#C4AE, 16#E4ED, 16#E4F6, 16#E4F4, 16#C2FE, 16#E4DD, 16#E4F0, 16#CAFE, 16#D5C4, 16#E4F1, 16#D1FA, 16#E4EB, 16#E4EC, 16#E4F2, 16#CEAB, 16#C5CB, 16#C7B1, 16#C2BA, 16#E4EA, 16#C1CA, 16#CCB6, 16#B3B1, 16#E4FB, 16#E4F3, 16#E4FA, 16#E4FD, 16#E4FC, 16#B3CE, 16#B3BA, 16#E4F7, 16#E4F9, 16#E4F8, 16#C5EC, 16#C0BD, 16#D4E8, 16#E5A2, 16#B0C4, 16#E5A4, 16#E5A3, 16#BCA4, 16#E5A5, 16#E5A1, 16#E4FE, 16#B1F4, 16#E5A8, 16#E5A9, 16#E5A6, 16#E5A7, 16#E5AA, 16#C6D9, 16#E5AB, 16#E5AD, 16#E5AC, 16#E5AF, 16#E5AE, 16#B9E0, 16#E5B0, 16#E5B1, 16#BBF0, 16#ECE1, 16#C3F0, 16#B5C6, 16#BBD2, 16#C1E9, 16#D4EE, 16#BEC4, 16#D7C6, 16#D4D6, 16#B2D3, 16#ECBE, 16#EAC1, 16#C2AF, 16#B4B6, 16#D1D7, 16#B3B4, 16#C8B2, 16#BFBB, 16#ECC0, 16#D6CB, 16#ECBF, 16#ECC1, 16#ECC5, 16#BEE6, 16#CCBF, 16#C5DA, 16#BEBC, 16#ECC6, 16#B1FE, 16#ECC4, 16#D5A8, 16#B5E3, 16#ECC2, 16#C1B6, 16#B3E3, 16#ECC3, 16#CBB8, 16#C0C3, 16#CCFE, 16#C1D2, 16#ECC8, 16#BAE6, 16#C0D3, 16#D6F2, 16#D1CC, 16#BFBE, 16#B7B3, 16#C9D5, 16#ECC7, 16#BBE2, 16#CCCC, 16#BDFD, 16#C8C8, 16#CFA9, 16#CDE9, 16#C5EB, 16#B7E9, 16#D1C9, 16#BAB8, 16#ECC9, 16#ECCA, 16#BBC0, 16#ECCB, 16#ECE2, 16#B1BA, 16#B7D9, 16#BDB9, 16#ECCC, 16#D1E6, 16#ECCD, 16#C8BB, 16#ECD1, 16#ECD3, 16#BBCD, 16#BCE5, 16#ECCF, 16#C9B7, 16#C3BA, 16#ECE3, 16#D5D5, 16#ECD0, 16#D6F3, 16#ECD2, 16#ECCE, 16#ECD4, 16#ECD5, 16#C9BF, 16#CFA8, 16#D0DC, 16#D1AC, 16#C8DB, 16#ECD6, 16#CEF5, 16#CAEC, 16#ECDA, 16#ECD9, 16#B0BE, 16#ECD7, 16#ECD8, 16#ECE4, 16#C8BC, 16#C1C7, 16#ECDC, 16#D1E0, 16#ECDB, 16#D4EF, 16#ECDD, 16#DBC6, 16#ECDE, 16#B1AC, 16#ECDF, 16#ECE0, 16#D7A6, 16#C5C0, 16#EBBC, 16#B0AE, 16#BEF4, 16#B8B8, 16#D2AF, 16#B0D6, 16#B5F9, 16#D8B3, 16#CBAC, 16#E3DD, 16#C6AC, 16#B0E6, 16#C5C6, 16#EBB9, 16#EBBA, 16#EBBB, 16#D1C0, 16#C5A3, 16#EAF2, 16#C4B2, 16#C4B5, 16#C0CE, 16#EAF3, 16#C4C1, 16#CEEF, 16#EAF0, 16#EAF4, 16#C9FC, 16#C7A3, 16#CCD8, 16#CEFE, 16#EAF5, 16#EAF6, 16#CFAC, 16#C0E7, 16#EAF7, 16#B6BF, 16#EAF8, 16#EAF9, 16#EAFA, 16#EAFB, 16#EAF1, 16#C8AE, 16#E1EB, 16#B7B8, 16#E1EC, 16#E1ED, 16#D7B4, 16#E1EE, 16#E1EF, 16#D3CC, 16#E1F1, 16#BFF1, 16#E1F0, 16#B5D2, 16#B1B7, 16#E1F3, 16#E1F2, 16#BAFC, 16#E1F4, 16#B9B7, 16#BED1, 16#C4FC, 16#BADD, 16#BDC6, 16#E1F5, 16#E1F7, 16#B6C0, 16#CFC1, 16#CAA8, 16#E1F6, 16#D5F8, 16#D3FC, 16#E1F8, 16#E1FC, 16#E1F9, 16#E1FA, 16#C0EA, 16#E1FE, 16#E2A1, 16#C0C7, 16#E1FB, 16#E1FD, 16#E2A5, 16#C1D4, 16#E2A3, 16#E2A8, 16#B2FE, 16#E2A2, 16#C3CD, 16#B2C2, 16#E2A7, 16#E2A6, 16#E2A4, 16#E2A9, 16#E2AB, 16#D0C9, 16#D6ED, 16#C3A8, 16#E2AC, 16#CFD7, 16#E2AE, 16#BAEF, 16#E9E0, 16#E2AD, 16#E2AA, 16#BBAB, 16#D4B3, 16#E2B0, 16#E2AF, 16#E9E1, 16#E2B1, 16#E2B2, 16#E2B3, 16#CCA1, 16#E2B4, 16#E2B5, 16#D0FE, 16#C2CA, 16#D3F1, 16#CDF5, 16#E7E0, 16#E7E1, 16#BEC1, 16#C2EA, 16#E7E4, 16#E7E3, 16#CDE6, 16#C3B5, 16#E7E2, 16#BBB7, 16#CFD6, 16#C1E1, 16#E7E9, 16#E7E8, 16#E7F4, 16#B2A3, 16#E7EA, 16#E7E6, 16#E7EC, 16#E7EB, 16#C9BA, 16#D5E4, 16#E7E5, 16#B7A9, 16#E7E7, 16#E7EE, 16#E7F3, 16#D6E9, 16#E7ED, 16#E7F2, 16#E7F1, 16#B0E0, 16#E7F5, 16#C7F2, 16#C0C5, 16#C0ED, 16#C1F0, 16#E7F0, 16#E7F6, 16#CBF6, 16#E8A2, 16#E8A1, 16#D7C1, 16#E7FA, 16#E7F9, 16#E7FB, 16#E7F7, 16#E7FE, 16#E7FD, 16#E7FC, 16#C1D5, 16#C7D9, 16#C5FD, 16#C5C3, 16#C7ED, 16#E8A3, 16#E8A6, 16#E8A5, 16#E8A7, 16#BAF7, 16#E7F8, 16#E8A4, 16#C8F0, 16#C9AA, 16#E8A9, 16#B9E5, 16#D1FE, 16#E8A8, 16#E8AA, 16#E8AD, 16#E8AE, 16#C1A7, 16#E8AF, 16#E8B0, 16#E8AC, 16#E8B4, 16#E8AB, 16#E8B1, 16#E8B5, 16#E8B2, 16#E8B3, 16#E8B7, 16#E8B6, 16#B9CF, 16#F0AC, 16#F0AD, 16#C6B0, 16#B0EA, 16#C8BF, 16#CDDF, 16#CECD, 16#EAB1, 16#EAB2, 16#C6BF, 16#B4C9, 16#EAB3, 16#D5E7, 16#DDF9, 16#EAB4, 16#EAB5, 16#EAB6, 16#B8CA, 16#DFB0, 16#C9F5, 16#CCF0, 16#C9FA, 16#C9FB, 16#D3C3, 16#CBA6, 16#B8A6, 16#F0AE, 16#B1C2, 16#E5B8, 16#CCEF, 16#D3C9, 16#BCD7, 16#C9EA, 16#B5E7, 16#C4D0, 16#B5E9, 16#EEAE, 16#BBAD, 16#E7DE, 16#EEAF, 16#B3A9, 16#EEB2, 16#EEB1, 16#BDE7, 16#EEB0, 16#CEB7, 16#C5CF, 16#C1F4, 16#DBCE, 16#EEB3, 16#D0F3, 16#C2D4, 16#C6E8, 16#B7AC, 16#EEB4, 16#B3EB, 16#BBFB, 16#EEB5, 16#E7DC, 16#EEB6, 16#BDAE, 16#F1E2, 16#CAE8, 16#D2C9, 16#F0DA, 16#F0DB, 16#F0DC, 16#C1C6, 16#B8ED, 16#BECE, 16#F0DE, 16#C5B1, 16#F0DD, 16#D1F1, 16#F0E0, 16#B0CC, 16#BDEA, 16#D2DF, 16#F0DF, 16#B4AF, 16#B7E8, 16#F0E6, 16#F0E5, 16#C6A3, 16#F0E1, 16#F0E2, 16#B4C3, 16#F0E3, 16#D5EE, 16#CCDB, 16#BED2, 16#BCB2, 16#F0E8, 16#F0E7, 16#F0E4, 16#B2A1, 16#D6A2, 16#D3B8, 16#BEB7, 16#C8AC, 16#F0EA, 16#D1F7, 16#D6CC, 16#BADB, 16#F0E9, 16#B6BB, 16#CDB4, 16#C6A6, 16#C1A1, 16#F0EB, 16#F0EE, 16#F0ED, 16#F0F0, 16#F0EC, 16#BBBE, 16#F0EF, 16#CCB5, 16#F0F2, 16#B3D5, 16#B1D4, 16#F0F3, 16#F0F4, 16#F0F6, 16#B4E1, 16#F0F1, 16#F0F7, 16#F0FA, 16#F0F8, 16#F0F5, 16#F0FD, 16#F0F9, 16#F0FC, 16#F0FE, 16#F1A1, 16#CEC1, 16#F1A4, 16#F1A3, 16#C1F6, 16#F0FB, 16#CADD, 16#B4F1, 16#B1F1, 16#CCB1, 16#F1A6, 16#F1A7, 16#F1AC, 16#D5CE, 16#F1A9, 16#C8B3, 16#F1A2, 16#F1AB, 16#F1A8, 16#F1A5, 16#F1AA, 16#B0A9, 16#F1AD, 16#F1AF, 16#F1B1, 16#F1B0, 16#F1AE, 16#D1A2, 16#F1B2, 16#F1B3, 16#B9EF, 16#B5C7, 16#B0D7, 16#B0D9, 16#D4ED, 16#B5C4, 16#BDD4, 16#BBCA, 16#F0A7, 16#B8DE, 16#F0A8, 16#B0A8, 16#F0A9, 16#CDEE, 16#F0AA, 16#F0AB, 16#C6A4, 16#D6E5, 16#F1E4, 16#F1E5, 16#C3F3, 16#D3DB, 16#D6D1, 16#C5E8, 16#D3AF, 16#D2E6, 16#EEC1, 16#B0BB, 16#D5B5, 16#D1CE, 16#BCE0, 16#BAD0, 16#BFF8, 16#B8C7, 16#B5C1, 16#C5CC, 16#CAA2, 16#C3CB, 16#EEC2, 16#C4BF, 16#B6A2, 16#EDEC, 16#C3A4, 16#D6B1, 16#CFE0, 16#EDEF, 16#C5CE, 16#B6DC, 16#CAA1, 16#EDED, 16#EDF0, 16#EDF1, 16#C3BC, 16#BFB4, 16#EDEE, 16#EDF4, 16#EDF2, 16#D5E6, 16#C3DF, 16#EDF3, 16#EDF6, 16#D5A3, 16#D1A3, 16#EDF5, 16#C3D0, 16#EDF7, 16#BFF4, 16#BEEC, 16#EDF8, 16#CCF7, 16#D1DB, 16#D7C5, 16#D5F6, 16#EDFC, 16#EDFB, 16#EDF9, 16#EDFA, 16#EDFD, 16#BEA6, 16#CBAF, 16#EEA1, 16#B6BD, 16#EEA2, 16#C4C0, 16#EDFE, 16#BDDE, 16#B2C7, 16#B6C3, 16#EEA5, 16#D8BA, 16#EEA3, 16#EEA6, 16#C3E9, 16#B3F2, 16#EEA7, 16#EEA4, 16#CFB9, 16#EEA8, 16#C2F7, 16#EEA9, 16#EEAA, 16#DEAB, 16#C6B3, 16#C7C6, 16#D6F5, 16#B5C9, 16#CBB2, 16#EEAB, 16#CDAB, 16#EEAC, 16#D5B0, 16#EEAD, 16#F6C4, 16#DBC7, 16#B4A3, 16#C3AC, 16#F1E6, 16#CAB8, 16#D2D3, 16#D6AA, 16#EFF2, 16#BED8, 16#BDC3, 16#EFF3, 16#B6CC, 16#B0AB, 16#CAAF, 16#EDB6, 16#EDB7, 16#CEF9, 16#B7AF, 16#BFF3, 16#EDB8, 16#C2EB, 16#C9B0, 16#EDB9, 16#C6F6, 16#BFB3, 16#EDBC, 16#C5F8, 16#D1D0, 16#D7A9, 16#EDBA, 16#EDBB, 16#D1E2, 16#EDBF, 16#EDC0, 16#EDC4, 16#EDC8, 16#EDC6, 16#EDCE, 16#D5E8, 16#EDC9, 16#EDC7, 16#EDBE, 16#C5E9, 16#C6C6, 16#C9E9, 16#D4D2, 16#EDC1, 16#EDC2, 16#EDC3, 16#EDC5, 16#C0F9, 16#B4A1, 16#B9E8, 16#EDD0, 16#EDD1, 16#EDCA, 16#EDCF, 16#CEF8, 16#CBB6, 16#EDCC, 16#EDCD, 16#CFF5, 16#EDD2, 16#C1F2, 16#D3B2, 16#EDCB, 16#C8B7, 16#BCEF, 16#C5F0, 16#EDD6, 16#B5EF, 16#C2B5, 16#B0AD, 16#CBE9, 16#B1AE, 16#EDD4, 16#CDEB, 16#B5E2, 16#EDD5, 16#EDD3, 16#EDD7, 16#B5FA, 16#EDD8, 16#EDD9, 16#EDDC, 16#B1CC, 16#C5F6, 16#BCEE, 16#EDDA, 16#CCBC, 16#B2EA, 16#EDDB, 16#C4EB, 16#B4C5, 16#B0F5, 16#EDDF, 16#C0DA, 16#B4E8, 16#C5CD, 16#EDDD, 16#BFC4, 16#EDDE, 16#C4A5, 16#EDE0, 16#EDE1, 16#EDE3, 16#C1D7, 16#BBC7, 16#BDB8, 16#EDE2, 16#EDE4, 16#EDE6, 16#EDE5, 16#EDE7, 16#CABE, 16#ECEA, 16#C0F1, 16#C9E7, 16#ECEB, 16#C6EE, 16#ECEC, 16#C6ED, 16#ECED, 16#ECF0, 16#D7E6, 16#ECF3, 16#ECF1, 16#ECEE, 16#ECEF, 16#D7A3, 16#C9F1, 16#CBEE, 16#ECF4, 16#ECF2, 16#CFE9, 16#ECF6, 16#C6B1, 16#BCC0, 16#ECF5, 16#B5BB, 16#BBF6, 16#ECF7, 16#D9F7, 16#BDFB, 16#C2BB, 16#ECF8, 16#ECF9, 16#B8A3, 16#ECFA, 16#ECFB, 16#ECFC, 16#D3ED, 16#D8AE, 16#C0EB, 16#C7DD, 16#BACC, 16#D0E3, 16#CBBD, 16#CDBA, 16#B8D1, 16#B1FC, 16#C7EF, 16#D6D6, 16#BFC6, 16#C3EB, 16#EFF5, 16#C3D8, 16#D7E2, 16#EFF7, 16#B3D3, 16#C7D8, 16#D1ED, 16#D6C8, 16#EFF8, 16#EFF6, 16#BBFD, 16#B3C6, 16#BDD5, 16#D2C6, 16#BBE0, 16#CFA1, 16#EFFC, 16#EFFB, 16#EFF9, 16#B3CC, 16#C9D4, 16#CBB0, 16#EFFE, 16#B0DE, 16#D6C9, 16#EFFD, 16#B3ED, 16#F6D5, 16#CEC8, 16#F0A2, 16#F0A1, 16#B5BE, 16#BCDA, 16#BBFC, 16#B8E5, 16#C4C2, 16#F0A3, 16#CBEB, 16#F0A6, 16#D1A8, 16#BEBF, 16#C7EE, 16#F1B6, 16#F1B7, 16#BFD5, 16#B4A9, 16#F1B8, 16#CDBB, 16#C7D4, 16#D5AD, 16#F1B9, 16#F1BA, 16#C7CF, 16#D2A4, 16#D6CF, 16#F1BB, 16#BDD1, 16#B4B0, 16#BEBD, 16#B4DC, 16#CED1, 16#BFDF, 16#F1BD, 16#BFFA, 16#F1BC, 16#F1BF, 16#F1BE, 16#F1C0, 16#F1C1, 16#C1FE, 16#C1A2, 16#CAFA, 16#D5BE, 16#BEBA, 16#BEB9, 16#D5C2, 16#BFA2, 16#CDAF, 16#F1B5, 16#BDDF, 16#B6CB, 16#D6F1, 16#F3C3, 16#F3C4, 16#B8CD, 16#F3C6, 16#F3C7, 16#B0CA, 16#F3C5, 16#F3C9, 16#CBF1, 16#F3CB, 16#D0A6, 16#B1CA, 16#F3C8, 16#F3CF, 16#B5D1, 16#F3D7, 16#F3D2, 16#F3D4, 16#F3D3, 16#B7FB, 16#B1BF, 16#F3CE, 16#F3CA, 16#B5DA, 16#F3D0, 16#F3D1, 16#F3D5, 16#F3CD, 16#BCE3, 16#C1FD, 16#F3D6, 16#F3DA, 16#F3CC, 16#B5C8, 16#BDEE, 16#F3DC, 16#B7A4, 16#BFF0, 16#D6FE, 16#CDB2, 16#B4F0, 16#B2DF, 16#F3D8, 16#F3D9, 16#C9B8, 16#F3DD, 16#F3DE, 16#F3E1, 16#F3DF, 16#F3E3, 16#F3E2, 16#F3DB, 16#BFEA, 16#B3EF, 16#F3E0, 16#C7A9, 16#BCF2, 16#F3EB, 16#B9BF, 16#F3E4, 16#B2AD, 16#BBFE, 16#CBE3, 16#F3ED, 16#F3E9, 16#B9DC, 16#F3EE, 16#F3E5, 16#F3E6, 16#F3EA, 16#C2E1, 16#F3EC, 16#F3EF, 16#F3E8, 16#BCFD, 16#CFE4, 16#F3F0, 16#F3E7, 16#F3F2, 16#D7AD, 16#C6AA, 16#F3F3, 16#F3F1, 16#C2A8, 16#B8DD, 16#F3F5, 16#F3F4, 16#B4DB, 16#F3F6, 16#F3F7, 16#F3F8, 16#C0BA, 16#C0E9, 16#C5F1, 16#F3FB, 16#F3FA, 16#B4D8, 16#F3FE, 16#F3F9, 16#F3FC, 16#F3FD, 16#F4A1, 16#F4A3, 16#BBC9, 16#F4A2, 16#F4A4, 16#B2BE, 16#F4A6, 16#F4A5, 16#BCAE, 16#C3D7, 16#D9E1, 16#C0E0, 16#F4CC, 16#D7D1, 16#B7DB, 16#F4CE, 16#C1A3, 16#C6C9, 16#B4D6, 16#D5B3, 16#F4D0, 16#F4CF, 16#F4D1, 16#CBDA, 16#F4D2, 16#D4C1, 16#D6E0, 16#B7E0, 16#C1B8, 16#C1BB, 16#F4D3, 16#BEAC, 16#B4E2, 16#F4D4, 16#F4D5, 16#BEAB, 16#F4D6, 16#F4DB, 16#F4D7, 16#F4DA, 16#BAFD, 16#F4D8, 16#F4D9, 16#B8E2, 16#CCC7, 16#F4DC, 16#B2DA, 16#C3D3, 16#D4E3, 16#BFB7, 16#F4DD, 16#C5B4, 16#F4E9, 16#CFB5, 16#CEC9, 16#CBD8, 16#CBF7, 16#BDF4, 16#D7CF, 16#C0DB, 16#D0F5, 16#F4EA, 16#F4EB, 16#F4EC, 16#F7E3, 16#B7B1, 16#F4ED, 16#D7EB, 16#F4EE, 16#E6F9, 16#BEC0, 16#E6FA, 16#BAEC, 16#E6FB, 16#CFCB, 16#E6FC, 16#D4BC, 16#BCB6, 16#E6FD, 16#E6FE, 16#BCCD, 16#C8D2, 16#CEB3, 16#E7A1, 16#B4BF, 16#E7A2, 16#C9B4, 16#B8D9, 16#C4C9, 16#D7DD, 16#C2DA, 16#B7D7, 16#D6BD, 16#CEC6, 16#B7C4, 16#C5A6, 16#E7A3, 16#CFDF, 16#E7A4, 16#E7A5, 16#E7A6, 16#C1B7, 16#D7E9, 16#C9F0, 16#CFB8, 16#D6AF, 16#D6D5, 16#E7A7, 16#B0ED, 16#E7A8, 16#E7A9, 16#C9DC, 16#D2EF, 16#BEAD, 16#E7AA, 16#B0F3, 16#C8DE, 16#BDE1, 16#E7AB, 16#C8C6, 16#E7AC, 16#BBE6, 16#B8F8, 16#D1A4, 16#E7AD, 16#C2E7, 16#BEF8, 16#BDCA, 16#CDB3, 16#E7AE, 16#E7AF, 16#BEEE, 16#D0E5, 16#CBE7, 16#CCD0, 16#BCCC, 16#E7B0, 16#BCA8, 16#D0F7, 16#E7B1, 16#D0F8, 16#E7B2, 16#E7B3, 16#B4C2, 16#E7B4, 16#E7B5, 16#C9FE, 16#CEAC, 16#C3E0, 16#E7B7, 16#B1C1, 16#B3F1, 16#E7B8, 16#E7B9, 16#D7DB, 16#D5C0, 16#E7BA, 16#C2CC, 16#D7BA, 16#E7BB, 16#E7BC, 16#E7BD, 16#BCEA, 16#C3E5, 16#C0C2, 16#E7BE, 16#E7BF, 16#BCA9, 16#E7C0, 16#E7C1, 16#E7B6, 16#B6D0, 16#E7C2, 16#E7C3, 16#E7C4, 16#BBBA, 16#B5DE, 16#C2C6, 16#B1E0, 16#E7C5, 16#D4B5, 16#E7C6, 16#B8BF, 16#E7C8, 16#E7C7, 16#B7EC, 16#E7C9, 16#B2F8, 16#E7CA, 16#E7CB, 16#E7CC, 16#E7CD, 16#E7CE, 16#E7CF, 16#E7D0, 16#D3A7, 16#CBF5, 16#E7D1, 16#E7D2, 16#E7D3, 16#E7D4, 16#C9C9, 16#E7D5, 16#E7D6, 16#E7D7, 16#E7D8, 16#E7D9, 16#BDC9, 16#E7DA, 16#F3BE, 16#B8D7, 16#C8B1, 16#F3BF, 16#F3C0, 16#F3C1, 16#B9DE, 16#CDF8, 16#D8E8, 16#BAB1, 16#C2DE, 16#EEB7, 16#B7A3, 16#EEB9, 16#EEB8, 16#B0D5, 16#EEBB, 16#D5D6, 16#D7EF, 16#D6C3, 16#EEBD, 16#CAF0, 16#EEBC, 16#EEBE, 16#EEC0, 16#EEBF, 16#D1F2, 16#C7BC, 16#C3C0, 16#B8E1, 16#C1E7, 16#F4C6, 16#D0DF, 16#F4C7, 16#CFDB, 16#C8BA, 16#F4C8, 16#F4C9, 16#F4CA, 16#F4CB, 16#D9FA, 16#B8FE, 16#E5F1, 16#D3F0, 16#F4E0, 16#CECC, 16#B3E1, 16#F1B4, 16#D2EE, 16#F4E1, 16#CFE8, 16#F4E2, 16#C7CC, 16#B5D4, 16#B4E4, 16#F4E4, 16#F4E3, 16#F4E5, 16#F4E6, 16#F4E7, 16#BAB2, 16#B0BF, 16#F4E8, 16#B7AD, 16#D2ED, 16#D2AB, 16#C0CF, 16#BFBC, 16#EBA3, 16#D5DF, 16#EAC8, 16#F1F3, 16#B6F8, 16#CBA3, 16#C4CD, 16#F1E7, 16#F1E8, 16#B8FB, 16#F1E9, 16#BAC4, 16#D4C5, 16#B0D2, 16#F1EA, 16#F1EB, 16#F1EC, 16#F1ED, 16#F1EE, 16#F1EF, 16#F1F1, 16#F1F0, 16#C5D5, 16#F1F2, 16#B6FA, 16#F1F4, 16#D2AE, 16#DEC7, 16#CBCA, 16#B3DC, 16#B5A2, 16#B9A2, 16#C4F4, 16#F1F5, 16#F1F6, 16#C1C4, 16#C1FB, 16#D6B0, 16#F1F7, 16#F1F8, 16#C1AA, 16#C6B8, 16#BEDB, 16#F1F9, 16#B4CF, 16#F1FA, 16#EDB2, 16#EDB1, 16#CBE0, 16#D2DE, 16#CBC1, 16#D5D8, 16#C8E2, 16#C0DF, 16#BCA1, 16#EBC1, 16#D0A4, 16#D6E2, 16#B6C7, 16#B8D8, 16#EBC0, 16#B8CE, 16#EBBF, 16#B3A6, 16#B9C9, 16#D6AB, 16#B7F4, 16#B7CA, 16#BCE7, 16#B7BE, 16#EBC6, 16#EBC7, 16#B0B9, 16#BFCF, 16#EBC5, 16#D3FD, 16#EBC8, 16#EBC9, 16#B7CE, 16#EBC2, 16#EBC4, 16#C9F6, 16#D6D7, 16#D5CD, 16#D0B2, 16#EBCF, 16#CEB8, 16#EBD0, 16#B5A8, 16#B1B3, 16#EBD2, 16#CCA5, 16#C5D6, 16#EBD3, 16#EBD1, 16#C5DF, 16#EBCE, 16#CAA4, 16#EBD5, 16#B0FB, 16#BAFA, 16#D8B7, 16#F1E3, 16#EBCA, 16#EBCB, 16#EBCC, 16#EBCD, 16#EBD6, 16#E6C0, 16#EBD9, 16#BFE8, 16#D2C8, 16#EBD7, 16#EBDC, 16#B8EC, 16#EBD8, 16#BDBA, 16#D0D8, 16#B0B7, 16#EBDD, 16#C4DC, 16#D6AC, 16#B4E0, 16#C2F6, 16#BCB9, 16#EBDA, 16#EBDB, 16#D4E0, 16#C6EA, 16#C4D4, 16#EBDF, 16#C5A7, 16#D9F5, 16#B2B1, 16#EBE4, 16#BDC5, 16#EBE2, 16#EBE3, 16#B8AC, 16#CDD1, 16#EBE5, 16#EBE1, 16#C1B3, 16#C6A2, 16#CCF3, 16#EBE6, 16#C0B0, 16#D2B8, 16#EBE7, 16#B8AF, 16#B8AD, 16#EBE8, 16#C7BB, 16#CDF3, 16#EBEA, 16#EBEB, 16#EBED, 16#D0C8, 16#EBF2, 16#EBEE, 16#EBF1, 16#C8F9, 16#D1FC, 16#EBEC, 16#EBE9, 16#B8B9, 16#CFD9, 16#C4E5, 16#EBEF, 16#EBF0, 16#CCDA, 16#CDC8, 16#B0F2, 16#EBF6, 16#EBF5, 16#B2B2, 16#B8E0, 16#EBF7, 16#B1EC, 16#CCC5, 16#C4A4, 16#CFA5, 16#EBF9, 16#ECA2, 16#C5F2, 16#EBFA, 16#C9C5, 16#E2DF, 16#EBFE, 16#CDCE, 16#ECA1, 16#B1DB, 16#D3B7, 16#D2DC, 16#EBFD, 16#EBFB, 16#B3BC, 16#EAB0, 16#D7D4, 16#F4AB, 16#B3F4, 16#D6C1, 16#D6C2, 16#D5E9, 16#BECA, 16#F4A7, 16#D2A8, 16#F4A8, 16#F4A9, 16#F4AA, 16#BECB, 16#D3DF, 16#C9E0, 16#C9E1, 16#F3C2, 16#CAE6, 16#CCF2, 16#E2B6, 16#CBB4, 16#CEE8, 16#D6DB, 16#F4AD, 16#F4AE, 16#F4AF, 16#F4B2, 16#BABD, 16#F4B3, 16#B0E3, 16#F4B0, 16#F4B1, 16#BDA2, 16#B2D5, 16#F4B6, 16#F4B7, 16#B6E6, 16#B2B0, 16#CFCF, 16#F4B4, 16#B4AC, 16#F4B5, 16#F4B8, 16#F4B9, 16#CDA7, 16#F4BA, 16#F4BB, 16#F4BC, 16#CBD2, 16#F4BD, 16#F4BE, 16#F4BF, 16#F4DE, 16#C1BC, 16#BCE8, 16#C9AB, 16#D1DE, 16#E5F5, 16#DCB3, 16#D2D5, 16#DCB4, 16#B0AC, 16#DCB5, 16#BDDA, 16#DCB9, 16#D8C2, 16#DCB7, 16#D3F3, 16#C9D6, 16#DCBA, 16#DCB6, 16#DCBB, 16#C3A2, 16#DCBC, 16#DCC5, 16#DCBD, 16#CEDF, 16#D6A5, 16#DCCF, 16#DCCD, 16#DCD2, 16#BDE6, 16#C2AB, 16#DCB8, 16#DCCB, 16#DCCE, 16#DCBE, 16#B7D2, 16#B0C5, 16#DCC7, 16#D0BE, 16#DCC1, 16#BBA8, 16#B7BC, 16#DCCC, 16#DCC6, 16#DCBF, 16#C7DB, 16#D1BF, 16#DCC0, 16#DCCA, 16#DCD0, 16#CEAD, 16#DCC2, 16#DCC3, 16#DCC8, 16#DCC9, 16#B2D4, 16#DCD1, 16#CBD5, 16#D4B7, 16#DCDB, 16#DCDF, 16#CCA6, 16#DCE6, 16#C3E7, 16#DCDC, 16#BFC1, 16#DCD9, 16#B0FA, 16#B9B6, 16#DCE5, 16#DCD3, 16#DCC4, 16#DCD6, 16#C8F4, 16#BFE0, 16#C9BB, 16#B1BD, 16#D3A2, 16#DCDA, 16#DCD5, 16#C6BB, 16#DCDE, 16#D7C2, 16#C3AF, 16#B7B6, 16#C7D1, 16#C3A9, 16#DCE2, 16#DCD8, 16#DCEB, 16#DCD4, 16#DCDD, 16#BEA5, 16#DCD7, 16#DCE0, 16#DCE3, 16#DCE4, 16#DCF8, 16#DCE1, 16#DDA2, 16#DCE7, 16#BCEB, 16#B4C4, 16#C3A3, 16#B2E7, 16#DCFA, 16#DCF2, 16#DCEF, 16#DCFC, 16#DCEE, 16#D2F0, 16#B2E8, 16#C8D7, 16#C8E3, 16#DCFB, 16#DCED, 16#DCF7, 16#DCF5, 16#BEA3, 16#DCF4, 16#B2DD, 16#DCF3, 16#BCF6, 16#DCE8, 16#BBC4, 16#C0F3, 16#BCD4, 16#DCE9, 16#DCEA, 16#DCF1, 16#DCF6, 16#DCF9, 16#B5B4, 16#C8D9, 16#BBE7, 16#DCFE, 16#DCFD, 16#D3AB, 16#DDA1, 16#DDA3, 16#DDA5, 16#D2F1, 16#DDA4, 16#DDA6, 16#DDA7, 16#D2A9, 16#BAC9, 16#DDA9, 16#DDB6, 16#DDB1, 16#DDB4, 16#DDB0, 16#C6CE, 16#C0F2, 16#C9AF, 16#DCEC, 16#DDAE, 16#DDB7, 16#DCF0, 16#DDAF, 16#DDB8, 16#DDAC, 16#DDB9, 16#DDB3, 16#DDAD, 16#C4AA, 16#DDA8, 16#C0B3, 16#C1AB, 16#DDAA, 16#DDAB, 16#DDB2, 16#BBF1, 16#DDB5, 16#D3A8, 16#DDBA, 16#DDBB, 16#C3A7, 16#DDD2, 16#DDBC, 16#DDD1, 16#B9BD, 16#BED5, 16#BEFA, 16#BACA, 16#DDCA, 16#DDC5, 16#DDBF, 16#B2CB, 16#DDC3, 16#DDCB, 16#B2A4, 16#DDD5, 16#DDBE, 16#C6D0, 16#DDD0, 16#DDD4, 16#C1E2, 16#B7C6, 16#DDCE, 16#DDCF, 16#DDC4, 16#DDBD, 16#DDCD, 16#CCD1, 16#DDC9, 16#DDC2, 16#C3C8, 16#C6BC, 16#CEAE, 16#DDCC, 16#DDC8, 16#DDC1, 16#DDC6, 16#C2DC, 16#D3A9, 16#D3AA, 16#DDD3, 16#CFF4, 16#C8F8, 16#DDE6, 16#DDC7, 16#DDE0, 16#C2E4, 16#DDE1, 16#DDD7, 16#D6F8, 16#DDD9, 16#DDD8, 16#B8F0, 16#DDD6, 16#C6CF, 16#B6AD, 16#DDE2, 16#BAF9, 16#D4E1, 16#DDE7, 16#B4D0, 16#DDDA, 16#BFFB, 16#DDE3, 16#DDDF, 16#DDDD, 16#B5D9, 16#DDDB, 16#DDDC, 16#DDDE, 16#BDAF, 16#DDE4, 16#DDE5, 16#DDF5, 16#C3C9, 16#CBE2, 16#DDF2, 16#D8E1, 16#C6D1, 16#DDF4, 16#D5F4, 16#DDF3, 16#DDF0, 16#DDEC, 16#DDEF, 16#DDE8, 16#D0EE, 16#C8D8, 16#DDEE, 16#DDE9, 16#DDEA, 16#CBF2, 16#DDED, 16#B1CD, 16#C0B6, 16#BCBB, 16#DDF1, 16#DDF7, 16#DDF6, 16#DDEB, 16#C5EE, 16#DDFB, 16#DEA4, 16#DEA3, 16#DDF8, 16#C3EF, 16#C2FB, 16#D5E1, 16#CEB5, 16#DDFD, 16#B2CC, 16#C4E8, 16#CADF, 16#C7BE, 16#DDFA, 16#DDFC, 16#DDFE, 16#DEA2, 16#B0AA, 16#B1CE, 16#DEAC, 16#DEA6, 16#BDB6, 16#C8EF, 16#DEA1, 16#DEA5, 16#DEA9, 16#DEA8, 16#DEA7, 16#DEAD, 16#D4CC, 16#DEB3, 16#DEAA, 16#DEAE, 16#C0D9, 16#B1A1, 16#DEB6, 16#DEB1, 16#DEB2, 16#D1A6, 16#DEB5, 16#DEAF, 16#DEB0, 16#D0BD, 16#DEB4, 16#CAED, 16#DEB9, 16#DEB8, 16#DEB7, 16#DEBB, 16#BDE5, 16#B2D8, 16#C3EA, 16#DEBA, 16#C5BA, 16#DEBC, 16#CCD9, 16#B7AA, 16#D4E5, 16#DEBD, 16#DEBF, 16#C4A2, 16#DEC1, 16#DEBE, 16#DEC0, 16#D5BA, 16#DEC2, 16#F2AE, 16#BBA2, 16#C2B2, 16#C5B0, 16#C2C7, 16#F2AF, 16#D0E9, 16#D3DD, 16#EBBD, 16#B3E6, 16#F2B0, 16#F2B1, 16#CAAD, 16#BAE7, 16#F2B3, 16#F2B5, 16#F2B4, 16#CBE4, 16#CFBA, 16#F2B2, 16#CAB4, 16#D2CF, 16#C2EC, 16#CEC3, 16#F2B8, 16#B0F6, 16#F2B7, 16#F2BE, 16#B2CF, 16#D1C1, 16#F2BA, 16#F2BC, 16#D4E9, 16#F2BB, 16#F2B6, 16#F2BF, 16#F2BD, 16#F2B9, 16#F2C7, 16#F2C4, 16#F2C6, 16#F2CA, 16#F2C2, 16#F2C0, 16#F2C5, 16#D6FB, 16#F2C1, 16#C7F9, 16#C9DF, 16#F2C8, 16#B9C6, 16#B5B0, 16#F2C3, 16#F2C9, 16#F2D0, 16#F2D6, 16#BBD7, 16#F2D5, 16#CDDC, 16#D6EB, 16#F2D2, 16#F2D4, 16#B8F2, 16#F2CB, 16#F2CE, 16#C2F9, 16#D5DD, 16#F2CC, 16#F2CD, 16#F2CF, 16#F2D3, 16#F2D9, 16#D3BC, 16#B6EA, 16#CAF1, 16#B7E4, 16#F2D7, 16#F2D8, 16#F2DA, 16#F2DD, 16#F2DB, 16#F2DC, 16#D1D1, 16#F2D1, 16#CDC9, 16#CECF, 16#D6A9, 16#F2E3, 16#C3DB, 16#F2E0, 16#C0AF, 16#F2EC, 16#F2DE, 16#F2E1, 16#F2E8, 16#F2E2, 16#F2E7, 16#F2E6, 16#F2E9, 16#F2DF, 16#F2E4, 16#F2EA, 16#D3AC, 16#F2E5, 16#B2F5, 16#F2F2, 16#D0AB, 16#F2F5, 16#BBC8, 16#F2F9, 16#F2F0, 16#F2F6, 16#F2F8, 16#F2FA, 16#F2F3, 16#F2F1, 16#BAFB, 16#B5FB, 16#F2EF, 16#F2F7, 16#F2ED, 16#F2EE, 16#F2EB, 16#F3A6, 16#F3A3, 16#F3A2, 16#F2F4, 16#C8DA, 16#F2FB, 16#F3A5, 16#C3F8, 16#F2FD, 16#F3A7, 16#F3A9, 16#F3A4, 16#F2FC, 16#F3AB, 16#F3AA, 16#C2DD, 16#F3AE, 16#F3B0, 16#F3A1, 16#F3B1, 16#F3AC, 16#F3AF, 16#F2FE, 16#F3AD, 16#F3B2, 16#F3B4, 16#F3A8, 16#F3B3, 16#F3B5, 16#D0B7, 16#F3B8, 16#D9F9, 16#F3B9, 16#F3B7, 16#C8E4, 16#F3B6, 16#F3BA, 16#F3BB, 16#B4C0, 16#EEC3, 16#F3BC, 16#F3BD, 16#D1AA, 16#F4AC, 16#D0C6, 16#D0D0, 16#D1DC, 16#CFCE, 16#BDD6, 16#D1C3, 16#BAE2, 16#E1E9, 16#D2C2, 16#F1C2, 16#B2B9, 16#B1ED, 16#F1C3, 16#C9C0, 16#B3C4, 16#D9F2, 16#CBA5, 16#F1C4, 16#D6D4, 16#F1C5, 16#F4C0, 16#F1C6, 16#D4AC, 16#F1C7, 16#B0C0, 16#F4C1, 16#F4C2, 16#B4FC, 16#C5DB, 16#CCBB, 16#D0E4, 16#CDE0, 16#F1C8, 16#D9F3, 16#B1BB, 16#CFAE, 16#B8A4, 16#F1CA, 16#F1CB, 16#B2C3, 16#C1D1, 16#D7B0, 16#F1C9, 16#F1CC, 16#F1CE, 16#D9F6, 16#D2E1, 16#D4A3, 16#F4C3, 16#C8B9, 16#F4C4, 16#F1CD, 16#F1CF, 16#BFE3, 16#F1D0, 16#F1D4, 16#F1D6, 16#F1D1, 16#C9D1, 16#C5E1, 16#C2E3, 16#B9FC, 16#F1D3, 16#F1D5, 16#B9D3, 16#F1DB, 16#BAD6, 16#B0FD, 16#F1D9, 16#F1D8, 16#F1D2, 16#F1DA, 16#F1D7, 16#C8EC, 16#CDCA, 16#F1DD, 16#E5BD, 16#F1DC, 16#F1DE, 16#F1DF, 16#CFE5, 16#F4C5, 16#BDF3, 16#F1E0, 16#F1E1, 16#CEF7, 16#D2AA, 16#F1FB, 16#B8B2, 16#BCFB, 16#B9DB, 16#B9E6, 16#C3D9, 16#CAD3, 16#EAE8, 16#C0C0, 16#BEF5, 16#EAE9, 16#EAEA, 16#EAEB, 16#EAEC, 16#EAED, 16#EAEE, 16#EAEF, 16#BDC7, 16#F5FB, 16#F5FD, 16#F5FE, 16#F5FC, 16#BDE2, 16#F6A1, 16#B4A5, 16#F6A2, 16#F6A3, 16#ECB2, 16#D1D4, 16#D9EA, 16#F6A4, 16#EEBA, 16#D5B2, 16#D3FE, 16#CCDC, 16#CAC4, 16#E5C0, 16#F6A5, 16#BEAF, 16#C6A9, 16#DAA5, 16#BCC6, 16#B6A9, 16#B8BC, 16#C8CF, 16#BCA5, 16#DAA6, 16#DAA7, 16#CCD6, 16#C8C3, 16#DAA8, 16#C6FD, 16#D1B5, 16#D2E9, 16#D1B6, 16#BCC7, 16#BDB2, 16#BBE4, 16#DAA9, 16#DAAA, 16#D1C8, 16#DAAB, 16#D0ED, 16#B6EF, 16#C2DB, 16#CBCF, 16#B7ED, 16#C9E8, 16#B7C3, 16#BEF7, 16#D6A4, 16#DAAC, 16#DAAD, 16#C6C0, 16#D7E7, 16#CAB6, 16#D5A9, 16#CBDF, 16#D5EF, 16#DAAE, 16#D6DF, 16#B4CA, 16#DAB0, 16#DAAF, 16#D2EB, 16#DAB1, 16#DAB2, 16#DAB3, 16#CAD4, 16#DAB4, 16#CAAB, 16#DAB5, 16#DAB6, 16#B3CF, 16#D6EF, 16#DAB7, 16#BBB0, 16#B5AE, 16#DAB8, 16#DAB9, 16#B9EE, 16#D1AF, 16#D2E8, 16#DABA, 16#B8C3, 16#CFEA, 16#B2EF, 16#DABB, 16#DABC, 16#BDEB, 16#CEDC, 16#D3EF, 16#DABD, 16#CEF3, 16#DABE, 16#D3D5, 16#BBE5, 16#DABF, 16#CBB5, 16#CBD0, 16#DAC0, 16#C7EB, 16#D6EE, 16#DAC1, 16#C5B5, 16#B6C1, 16#DAC2, 16#B7CC, 16#BFCE, 16#DAC3, 16#DAC4, 16#CBAD, 16#DAC5, 16#B5F7, 16#DAC6, 16#C1C2, 16#D7BB, 16#DAC7, 16#CCB8, 16#D2EA, 16#C4B1, 16#DAC8, 16#B5FD, 16#BBD1, 16#DAC9, 16#D0B3, 16#DACA, 16#DACB, 16#CEBD, 16#DACC, 16#DACD, 16#DACE, 16#B2F7, 16#DAD1, 16#DACF, 16#D1E8, 16#DAD0, 16#C3D5, 16#DAD2, 16#DAD3, 16#DAD4, 16#DAD5, 16#D0BB, 16#D2A5, 16#B0F9, 16#DAD6, 16#C7AB, 16#DAD7, 16#BDF7, 16#C3A1, 16#DAD8, 16#DAD9, 16#C3FD, 16#CCB7, 16#DADA, 16#DADB, 16#C0BE, 16#C6D7, 16#DADC, 16#DADD, 16#C7B4, 16#DADE, 16#DADF, 16#B9C8, 16#BBED, 16#B6B9, 16#F4F8, 16#F4F9, 16#CDE3, 16#F5B9, 16#EBE0, 16#CFF3, 16#BBBF, 16#BAC0, 16#D4A5, 16#E1D9, 16#F5F4, 16#B1AA, 16#B2F2, 16#F5F5, 16#F5F7, 16#BAD1, 16#F5F6, 16#C3B2, 16#F5F9, 16#F5F8, 16#B1B4, 16#D5EA, 16#B8BA, 16#B9B1, 16#B2C6, 16#D4F0, 16#CFCD, 16#B0DC, 16#D5CB, 16#BBF5, 16#D6CA, 16#B7B7, 16#CCB0, 16#C6B6, 16#B1E1, 16#B9BA, 16#D6FC, 16#B9E1, 16#B7A1, 16#BCFA, 16#EADA, 16#EADB, 16#CCF9, 16#B9F3, 16#EADC, 16#B4FB, 16#C3B3, 16#B7D1, 16#BAD8, 16#EADD, 16#D4F4, 16#EADE, 16#BCD6, 16#BBDF, 16#EADF, 16#C1DE, 16#C2B8, 16#D4DF, 16#D7CA, 16#EAE0, 16#EAE1, 16#EAE4, 16#EAE2, 16#EAE3, 16#C9DE, 16#B8B3, 16#B6C4, 16#EAE5, 16#CAEA, 16#C9CD, 16#B4CD, 16#E2D9, 16#C5E2, 16#EAE6, 16#C0B5, 16#D7B8, 16#EAE7, 16#D7AC, 16#C8FC, 16#D8D3, 16#D8CD, 16#D4DE, 16#D4F9, 16#C9C4, 16#D3AE, 16#B8D3, 16#B3E0, 16#C9E2, 16#F4F6, 16#BAD5, 16#F4F7, 16#D7DF, 16#F4F1, 16#B8B0, 16#D5D4, 16#B8CF, 16#C6F0, 16#B3C3, 16#F4F2, 16#B3AC, 16#D4BD, 16#C7F7, 16#F4F4, 16#F4F3, 16#CCCB, 16#C8A4, 16#F4F5, 16#D7E3, 16#C5BF, 16#F5C0, 16#F5BB, 16#F5C3, 16#F5C2, 16#D6BA, 16#F5C1, 16#D4BE, 16#F5C4, 16#F5CC, 16#B0CF, 16#B5F8, 16#F5C9, 16#F5CA, 16#C5DC, 16#F5C5, 16#F5C6, 16#F5C7, 16#F5CB, 16#BEE0, 16#F5C8, 16#B8FA, 16#F5D0, 16#F5D3, 16#BFE7, 16#B9F2, 16#F5BC, 16#F5CD, 16#C2B7, 16#CCF8, 16#BCF9, 16#F5CE, 16#F5CF, 16#F5D1, 16#B6E5, 16#F5D2, 16#F5D5, 16#F5BD, 16#F5D4, 16#D3BB, 16#B3EC, 16#CCA4, 16#F5D6, 16#F5D7, 16#BEE1, 16#F5D8, 16#CCDF, 16#F5DB, 16#B2C8, 16#D7D9, 16#F5D9, 16#F5DA, 16#F5DC, 16#F5E2, 16#F5E0, 16#F5DF, 16#F5DD, 16#F5E1, 16#F5DE, 16#F5E4, 16#F5E5, 16#CCE3, 16#E5BF, 16#B5B8, 16#F5E3, 16#F5E8, 16#CCA3, 16#F5E6, 16#F5E7, 16#F5BE, 16#B1C4, 16#F5BF, 16#B5C5, 16#B2E4, 16#F5EC, 16#F5E9, 16#B6D7, 16#F5ED, 16#F5EA, 16#F5EB, 16#B4DA, 16#D4EA, 16#F5EE, 16#B3F9, 16#F5EF, 16#F5F1, 16#F5F0, 16#F5F2, 16#F5F3, 16#C9ED, 16#B9AA, 16#C7FB, 16#B6E3, 16#CCC9, 16#EAA6, 16#B3B5, 16#D4FE, 16#B9EC, 16#D0F9, 16#E9ED, 16#D7AA, 16#E9EE, 16#C2D6, 16#C8ED, 16#BAE4, 16#E9EF, 16#E9F0, 16#E9F1, 16#D6E1, 16#E9F2, 16#E9F3, 16#E9F5, 16#E9F4, 16#E9F6, 16#E9F7, 16#C7E1, 16#E9F8, 16#D4D8, 16#E9F9, 16#BDCE, 16#E9FA, 16#E9FB, 16#BDCF, 16#E9FC, 16#B8A8, 16#C1BE, 16#E9FD, 16#B1B2, 16#BBD4, 16#B9F5, 16#E9FE, 16#EAA1, 16#EAA2, 16#EAA3, 16#B7F8, 16#BCAD, 16#CAE4, 16#E0CE, 16#D4AF, 16#CFBD, 16#D5B7, 16#EAA4, 16#D5DE, 16#EAA5, 16#D0C1, 16#B9BC, 16#B4C7, 16#B1D9, 16#C0B1, 16#B1E6, 16#B1E7, 16#B1E8, 16#B3BD, 16#C8E8, 16#E5C1, 16#B1DF, 16#C1C9, 16#B4EF, 16#C7A8, 16#D3D8, 16#C6F9, 16#D1B8, 16#B9FD, 16#C2F5, 16#D3AD, 16#D4CB, 16#BDFC, 16#E5C2, 16#B7B5, 16#E5C3, 16#BBB9, 16#D5E2, 16#BDF8, 16#D4B6, 16#CEA5, 16#C1AC, 16#B3D9, 16#CCF6, 16#E5C6, 16#E5C4, 16#E5C8, 16#E5CA, 16#E5C7, 16#B5CF, 16#C6C8, 16#B5FC, 16#E5C5, 16#CAF6, 16#E5C9, 16#C3D4, 16#B1C5, 16#BCA3, 16#D7B7, 16#CDCB, 16#CBCD, 16#CACA, 16#CCD3, 16#E5CC, 16#E5CB, 16#C4E6, 16#D1A1, 16#D1B7, 16#E5CD, 16#E5D0, 16#CDB8, 16#D6F0, 16#E5CF, 16#B5DD, 16#CDBE, 16#E5D1, 16#B6BA, 16#CDA8, 16#B9E4, 16#CAC5, 16#B3D1, 16#CBD9, 16#D4EC, 16#E5D2, 16#B7EA, 16#E5CE, 16#E5D5, 16#B4FE, 16#E5D6, 16#E5D3, 16#E5D4, 16#D2DD, 16#C2DF, 16#B1C6, 16#D3E2, 16#B6DD, 16#CBEC, 16#E5D7, 16#D3F6, 16#B1E9, 16#B6F4, 16#E5DA, 16#E5D8, 16#E5D9, 16#B5C0, 16#D2C5, 16#E5DC, 16#E5DE, 16#E5DD, 16#C7B2, 16#D2A3, 16#E5DB, 16#D4E2, 16#D5DA, 16#E5E0, 16#D7F1, 16#E5E1, 16#B1DC, 16#D1FB, 16#E5E2, 16#E5E4, 16#E5E3, 16#E5E5, 16#D2D8, 16#B5CB, 16#E7DF, 16#DAF5, 16#DAF8, 16#DAF6, 16#DAF7, 16#DAFA, 16#D0CF, 16#C4C7, 16#B0EE, 16#D0B0, 16#DAF9, 16#D3CA, 16#BAAA, 16#DBA2, 16#C7F1, 16#DAFC, 16#DAFB, 16#C9DB, 16#DAFD, 16#DBA1, 16#D7DE, 16#DAFE, 16#C1DA, 16#DBA5, 16#D3F4, 16#DBA7, 16#DBA4, 16#DBA8, 16#BDBC, 16#C0C9, 16#DBA3, 16#DBA6, 16#D6A3, 16#DBA9, 16#DBAD, 16#DBAE, 16#DBAC, 16#BAC2, 16#BFA4, 16#DBAB, 16#DBAA, 16#D4C7, 16#B2BF, 16#DBAF, 16#B9F9, 16#DBB0, 16#B3BB, 16#B5A6, 16#B6BC, 16#DBB1, 16#B6F5, 16#DBB2, 16#B1C9, 16#DBB4, 16#DBB3, 16#DBB5, 16#DBB7, 16#DBB6, 16#DBB8, 16#DBB9, 16#DBBA, 16#D3CF, 16#F4FA, 16#C7F5, 16#D7C3, 16#C5E4, 16#F4FC, 16#F4FD, 16#F4FB, 16#BEC6, 16#D0EF, 16#B7D3, 16#D4CD, 16#CCAA, 16#F5A2, 16#F5A1, 16#BAA8, 16#F4FE, 16#CBD6, 16#F5A4, 16#C0D2, 16#B3EA, 16#CDAA, 16#F5A5, 16#F5A3, 16#BDB4, 16#F5A8, 16#F5A9, 16#BDCD, 16#C3B8, 16#BFE1, 16#CBE1, 16#F5AA, 16#F5A6, 16#F5A7, 16#C4F0, 16#F5AC, 16#B4BC, 16#D7ED, 16#B4D7, 16#F5AB, 16#F5AE, 16#F5AD, 16#F5AF, 16#D0D1, 16#C3D1, 16#C8A9, 16#F5B0, 16#F5B1, 16#F5B2, 16#F5B3, 16#F5B4, 16#F5B5, 16#F5B7, 16#F5B6, 16#F5B8, 16#B2C9, 16#D3D4, 16#CACD, 16#C0EF, 16#D6D8, 16#D2B0, 16#C1BF, 16#BDF0, 16#B8AA, 16#BCF8, 16#F6C6, 16#F6C7, 16#F6C8, 16#F6C9, 16#F6CA, 16#F6CC, 16#F6CB, 16#F7E9, 16#F6CD, 16#F6CE, 16#EEC4, 16#EEC5, 16#EEC6, 16#D5EB, 16#B6A4, 16#EEC8, 16#EEC7, 16#EEC9, 16#EECA, 16#C7A5, 16#EECB, 16#EECC, 16#B7B0, 16#B5F6, 16#EECD, 16#EECF, 16#EECE, 16#B8C6, 16#EED0, 16#EED1, 16#EED2, 16#B6DB, 16#B3AE, 16#D6D3, 16#C4C6, 16#B1B5, 16#B8D6, 16#EED3, 16#EED4, 16#D4BF, 16#C7D5, 16#BEFB, 16#CED9, 16#B9B3, 16#EED6, 16#EED5, 16#EED8, 16#EED7, 16#C5A5, 16#EED9, 16#EEDA, 16#C7AE, 16#EEDB, 16#C7AF, 16#EEDC, 16#B2A7, 16#EEDD, 16#EEDE, 16#EEDF, 16#EEE0, 16#EEE1, 16#D7EA, 16#EEE2, 16#EEE3, 16#BCD8, 16#EEE4, 16#D3CB, 16#CCFA, 16#B2AC, 16#C1E5, 16#EEE5, 16#C7A6, 16#C3AD, 16#EEE6, 16#EEE7, 16#EEE8, 16#EEE9, 16#EEEA, 16#EEEB, 16#EEEC, 16#EEED, 16#EEEE, 16#EEEF, 16#EEF0, 16#EEF1, 16#EEF2, 16#EEF4, 16#EEF3, 16#EEF5, 16#CDAD, 16#C2C1, 16#EEF6, 16#EEF7, 16#EEF8, 16#D5A1, 16#EEF9, 16#CFB3, 16#EEFA, 16#EEFB, 16#EEFC, 16#EEFD, 16#EFA1, 16#EEFE, 16#EFA2, 16#B8F5, 16#C3FA, 16#EFA3, 16#EFA4, 16#BDC2, 16#D2BF, 16#B2F9, 16#EFA5, 16#EFA6, 16#EFA7, 16#D2F8, 16#EFA8, 16#D6FD, 16#EFA9, 16#C6CC, 16#EFAA, 16#EFAB, 16#C1B4, 16#EFAC, 16#CFFA, 16#CBF8, 16#EFAE, 16#EFAD, 16#B3FA, 16#B9F8, 16#EFAF, 16#EFB0, 16#D0E2, 16#EFB1, 16#EFB2, 16#B7E6, 16#D0BF, 16#EFB3, 16#EFB4, 16#EFB5, 16#C8F1, 16#CCE0, 16#EFB6, 16#EFB7, 16#EFB8, 16#EFB9, 16#EFBA, 16#D5E0, 16#EFBB, 16#B4ED, 16#C3AA, 16#EFBC, 16#EFBD, 16#EFBE, 16#EFBF, 16#CEFD, 16#EFC0, 16#C2E0, 16#B4B8, 16#D7B6, 16#BDF5, 16#CFC7, 16#EFC3, 16#EFC1, 16#EFC2, 16#EFC4, 16#B6A7, 16#BCFC, 16#BEE2, 16#C3CC, 16#EFC5, 16#EFC6, 16#EFC7, 16#EFCF, 16#EFC8, 16#EFC9, 16#EFCA, 16#C7C2, 16#EFF1, 16#B6CD, 16#EFCB, 16#EFCC, 16#EFCD, 16#B6C6, 16#C3BE, 16#EFCE, 16#EFD0, 16#EFD1, 16#EFD2, 16#D5F2, 16#EFD3, 16#C4F7, 16#EFD4, 16#C4F8, 16#EFD5, 16#EFD6, 16#B8E4, 16#B0F7, 16#EFD7, 16#EFD8, 16#EFD9, 16#EFDA, 16#EFDB, 16#EFDC, 16#EFDD, 16#EFDE, 16#BEB5, 16#EFE1, 16#EFDF, 16#EFE0, 16#EFE2, 16#EFE3, 16#C1CD, 16#EFE4, 16#EFE5, 16#EFE6, 16#EFE7, 16#EFE8, 16#EFE9, 16#EFEA, 16#EFEB, 16#EFEC, 16#C0D8, 16#EFED, 16#C1AD, 16#EFEE, 16#EFEF, 16#EFF0, 16#CFE2, 16#B3A4, 16#C3C5, 16#E3C5, 16#C9C1, 16#E3C6, 16#B1D5, 16#CECA, 16#B4B3, 16#C8F2, 16#E3C7, 16#CFD0, 16#E3C8, 16#BCE4, 16#E3C9, 16#E3CA, 16#C3C6, 16#D5A2, 16#C4D6, 16#B9EB, 16#CEC5, 16#E3CB, 16#C3F6, 16#E3CC, 16#B7A7, 16#B8F3, 16#BAD2, 16#E3CD, 16#E3CE, 16#D4C4, 16#E3CF, 16#E3D0, 16#D1CB, 16#E3D1, 16#E3D2, 16#E3D3, 16#E3D4, 16#D1D6, 16#E3D5, 16#B2FB, 16#C0BB, 16#E3D6, 16#C0AB, 16#E3D7, 16#E3D8, 16#E3D9, 16#E3DA, 16#E3DB, 16#B8B7, 16#DAE2, 16#B6D3, 16#DAE4, 16#DAE3, 16#DAE6, 16#C8EE, 16#DAE5, 16#B7C0, 16#D1F4, 16#D2F5, 16#D5F3, 16#BDD7, 16#D7E8, 16#DAE8, 16#DAE7, 16#B0A2, 16#CDD3, 16#DAE9, 16#B8BD, 16#BCCA, 16#C2BD, 16#C2A4, 16#B3C2, 16#DAEA, 16#C2AA, 16#C4B0, 16#BDB5, 16#CFDE, 16#DAEB, 16#C9C2, 16#B1DD, 16#DAEC, 16#B6B8, 16#D4BA, 16#B3FD, 16#DAED, 16#D4C9, 16#CFD5, 16#C5E3, 16#DAEE, 16#DAEF, 16#DAF0, 16#C1EA, 16#CCD5, 16#CFDD, 16#D3E7, 16#C2A1, 16#DAF1, 16#CBE5, 16#DAF2, 16#CBE6, 16#D2FE, 16#B8F4, 16#DAF3, 16#B0AF, 16#CFB6, 16#D5CF, 16#CBED, 16#DAF4, 16#E3C4, 16#C1A5, 16#F6BF, 16#F6C0, 16#F6C1, 16#C4D1, 16#C8B8, 16#D1E3, 16#D0DB, 16#D1C5, 16#BCAF, 16#B9CD, 16#EFF4, 16#B4C6, 16#D3BA, 16#F6C2, 16#B3FB, 16#F6C3, 16#B5F1, 16#F6C5, 16#D3EA, 16#F6A7, 16#D1A9, 16#F6A9, 16#F6A8, 16#C1E3, 16#C0D7, 16#B1A2, 16#CEED, 16#D0E8, 16#F6AB, 16#CFF6, 16#F6AA, 16#D5F0, 16#F6AC, 16#C3B9, 16#BBF4, 16#F6AE, 16#F6AD, 16#C4DE, 16#C1D8, 16#CBAA, 16#CFBC, 16#F6AF, 16#F6B0, 16#F6B1, 16#C2B6, 16#B0D4, 16#C5F9, 16#F6B2, 16#C7E0, 16#F6A6, 16#BEB8, 16#BEB2, 16#B5E5, 16#B7C7, 16#BFBF, 16#C3D2, 16#C3E6, 16#D8CC, 16#B8EF, 16#BDF9, 16#D1A5, 16#B0D0, 16#F7B0, 16#F7B1, 16#D0AC, 16#B0B0, 16#F7B2, 16#F7B3, 16#F7B4, 16#C7CA, 16#BECF, 16#F7B7, 16#F7B6, 16#B1DE, 16#F7B5, 16#F7B8, 16#F7B9, 16#CEA4, 16#C8CD, 16#BAAB, 16#E8B8, 16#E8B9, 16#E8BA, 16#BEC2, 16#D2F4, 16#D4CF, 16#C9D8, 16#D2B3, 16#B6A5, 16#C7EA, 16#F1FC, 16#CFEE, 16#CBB3, 16#D0EB, 16#E7EF, 16#CDE7, 16#B9CB, 16#B6D9, 16#F1FD, 16#B0E4, 16#CBCC, 16#F1FE, 16#D4A4, 16#C2AD, 16#C1EC, 16#C6C4, 16#BEB1, 16#F2A1, 16#BCD5, 16#F2A2, 16#F2A3, 16#F2A4, 16#D2C3, 16#C6B5, 16#CDC7, 16#F2A5, 16#D3B1, 16#BFC5, 16#CCE2, 16#F2A6, 16#F2A7, 16#D1D5, 16#B6EE, 16#F2A8, 16#F2A9, 16#B5DF, 16#F2AA, 16#F2AB, 16#B2FC, 16#F2AC, 16#F2AD, 16#C8A7, 16#B7E7, 16#ECA9, 16#ECAA, 16#ECAB, 16#ECAC, 16#C6AE, 16#ECAD, 16#ECAE, 16#B7C9, 16#CAB3, 16#E2B8, 16#F7CF, 16#F7D0, 16#B2CD, 16#F7D1, 16#F7D3, 16#F7D2, 16#E2BB, 16#BCA2, 16#E2BC, 16#E2BD, 16#E2BE, 16#E2BF, 16#E2C0, 16#E2C1, 16#B7B9, 16#D2FB, 16#BDA4, 16#CACE, 16#B1A5, 16#CBC7, 16#E2C2, 16#B6FC, 16#C8C4, 16#E2C3, 16#BDC8, 16#B1FD, 16#E2C4, 16#B6F6, 16#E2C5, 16#C4D9, 16#E2C6, 16#CFDA, 16#B9DD, 16#E2C7, 16#C0A1, 16#E2C8, 16#B2F6, 16#E2C9, 16#C1F3, 16#E2CA, 16#E2CB, 16#C2F8, 16#E2CC, 16#E2CD, 16#E2CE, 16#CAD7, 16#D8B8, 16#D9E5, 16#CFE3, 16#F0A5, 16#DCB0, 16#C2ED, 16#D4A6, 16#CDD4, 16#D1B1, 16#B3DB, 16#C7FD, 16#B2B5, 16#C2BF, 16#E6E0, 16#CABB, 16#E6E1, 16#E6E2, 16#BED4, 16#E6E3, 16#D7A4, 16#CDD5, 16#E6E5, 16#BCDD, 16#E6E4, 16#E6E6, 16#E6E7, 16#C2EE, 16#BDBE, 16#E6E8, 16#C2E6, 16#BAA7, 16#E6E9, 16#E6EA, 16#B3D2, 16#D1E9, 16#BFA5, 16#E6EB, 16#C6EF, 16#E6EC, 16#E6ED, 16#E6EE, 16#C6AD, 16#E6EF, 16#C9A7, 16#E6F0, 16#E6F1, 16#E6F2, 16#E5B9, 16#E6F3, 16#E6F4, 16#C2E2, 16#E6F5, 16#E6F6, 16#D6E8, 16#E6F7, 16#E6F8, 16#B9C7, 16#F7BB, 16#F7BA, 16#F7BE, 16#F7BC, 16#BAA1, 16#F7BF, 16#F7C0, 16#F7C2, 16#F7C1, 16#F7C4, 16#F7C3, 16#F7C5, 16#F7C6, 16#F7C7, 16#CBE8, 16#B8DF, 16#F7D4, 16#F7D5, 16#F7D6, 16#F7D8, 16#F7DA, 16#F7D7, 16#F7DB, 16#F7D9, 16#D7D7, 16#F7DC, 16#F7DD, 16#F7DE, 16#F7DF, 16#F7E0, 16#DBCB, 16#D8AA, 16#E5F7, 16#B9ED, 16#BFFD, 16#BBEA, 16#F7C9, 16#C6C7, 16#F7C8, 16#F7CA, 16#F7CC, 16#F7CB, 16#F7CD, 16#CEBA, 16#F7CE, 16#C4A7, 16#D3E3, 16#F6CF, 16#C2B3, 16#F6D0, 16#F6D1, 16#F6D2, 16#F6D3, 16#F6D4, 16#F6D6, 16#B1AB, 16#F6D7, 16#F6D8, 16#F6D9, 16#F6DA, 16#F6DB, 16#F6DC, 16#F6DD, 16#F6DE, 16#CFCA, 16#F6DF, 16#F6E0, 16#F6E1, 16#F6E2, 16#F6E3, 16#F6E4, 16#C0F0, 16#F6E5, 16#F6E6, 16#F6E7, 16#F6E8, 16#F6E9, 16#F6EA, 16#F6EB, 16#F6EC, 16#F6ED, 16#F6EE, 16#F6EF, 16#F6F0, 16#F6F1, 16#F6F2, 16#F6F3, 16#F6F4, 16#BEA8, 16#F6F5, 16#F6F6, 16#F6F7, 16#F6F8, 16#C8FA, 16#F6F9, 16#F6FA, 16#F6FB, 16#F6FC, 16#F6FD, 16#F6FE, 16#F7A1, 16#F7A2, 16#F7A3, 16#F7A4, 16#F7A5, 16#F7A6, 16#F7A7, 16#F7A8, 16#B1EE, 16#F7A9, 16#F7AA, 16#F7AB, 16#F7AC, 16#F7AD, 16#C1DB, 16#F7AE, 16#F7AF, 16#C4F1, 16#F0AF, 16#BCA6, 16#F0B0, 16#C3F9, 16#C5B8, 16#D1BB, 16#F0B1, 16#F0B2, 16#F0B3, 16#F0B4, 16#F0B5, 16#D1BC, 16#D1EC, 16#F0B7, 16#F0B6, 16#D4A7, 16#CDD2, 16#F0B8, 16#F0BA, 16#F0B9, 16#F0BB, 16#F0BC, 16#B8EB, 16#F0BD, 16#BAE8, 16#F0BE, 16#F0BF, 16#BEE9, 16#F0C0, 16#B6EC, 16#F0C1, 16#F0C2, 16#F0C3, 16#F0C4, 16#C8B5, 16#F0C5, 16#F0C6, 16#F0C7, 16#C5F4, 16#F0C8, 16#F0C9, 16#F0CA, 16#F7BD, 16#F0CB, 16#F0CC, 16#F0CD, 16#F0CE, 16#F0CF, 16#BAD7, 16#F0D0, 16#F0D1, 16#F0D2, 16#F0D3, 16#F0D4, 16#F0D5, 16#F0D6, 16#F0D8, 16#D3A5, 16#F0D7, 16#F0D9, 16#F5BA, 16#C2B9, 16#F7E4, 16#F7E5, 16#F7E6, 16#F7E7, 16#F7E8, 16#C2B4, 16#F7EA, 16#F7EB, 16#C2F3, 16#F4F0, 16#F4EF, 16#C2E9, 16#F7E1, 16#F7E2, 16#BBC6, 16#D9E4, 16#CAF2, 16#C0E8, 16#F0A4, 16#BADA, 16#C7AD, 16#C4AC, 16#F7EC, 16#F7ED, 16#F7EE, 16#F7F0, 16#F7EF, 16#F7F1, 16#F7F4, 16#F7F3, 16#F7F2, 16#F7F5, 16#F7F6, 16#EDE9, 16#EDEA, 16#EDEB, 16#F6BC, 16#F6BD, 16#F6BE, 16#B6A6, 16#D8BE, 16#B9C4, 16#D8BB, 16#DCB1, 16#CAF3, 16#F7F7, 16#F7F8, 16#F7F9, 16#F7FB, 16#F7FA, 16#B1C7, 16#F7FC, 16#F7FD, 16#F7FE, 16#C6EB, 16#ECB4, 16#B3DD, 16#F6B3, 16#F6B4, 16#C1E4, 16#F6B5, 16#F6B6, 16#F6B7, 16#F6B8, 16#F6B9, 16#F6BA, 16#C8A3, 16#F6BB, 16#C1FA, 16#B9A8, 16#EDE8, 16#B9EA, 16#D9DF, 16#A6F2, 16#A6F4, 16#A6F5, 16#A6E0, 16#A6E1, 16#A6F0, 16#A6F1, 16#A6E2, 16#A6E3, 16#A6EE, 16#A6EF, 16#A6E6, 16#A6E7, 16#A6E4, 16#A6E5, 16#A6E8, 16#A6E9, 16#A6EA, 16#A6EB, 16#A3A1, 16#A3A2, 16#A3A3, 16#A1E7, 16#A3A5, 16#A3A6, 16#A3A7, 16#A3A8, 16#A3A9, 16#A3AA, 16#A3AB, 16#A3AC, 16#A3AD, 16#A3AE, 16#A3AF, 16#A3B0, 16#A3B1, 16#A3B2, 16#A3B3, 16#A3B4, 16#A3B5, 16#A3B6, 16#A3B7, 16#A3B8, 16#A3B9, 16#A3BA, 16#A3BB, 16#A3BC, 16#A3BD, 16#A3BE, 16#A3BF, 16#A3C0, 16#A3C1, 16#A3C2, 16#A3C3, 16#A3C4, 16#A3C5, 16#A3C6, 16#A3C7, 16#A3C8, 16#A3C9, 16#A3CA, 16#A3CB, 16#A3CC, 16#A3CD, 16#A3CE, 16#A3CF, 16#A3D0, 16#A3D1, 16#A3D2, 16#A3D3, 16#A3D4, 16#A3D5, 16#A3D6, 16#A3D7, 16#A3D8, 16#A3D9, 16#A3DA, 16#A3DB, 16#A3DC, 16#A3DD, 16#A3DE, 16#A3DF, 16#A3E0, 16#A3E1, 16#A3E2, 16#A3E3, 16#A3E4, 16#A3E5, 16#A3E6, 16#A3E7, 16#A3E8, 16#A3E9, 16#A3EA, 16#A3EB, 16#A3EC, 16#A3ED, 16#A3EE, 16#A3EF, 16#A3F0, 16#A3F1, 16#A3F2, 16#A3F3, 16#A3F4, 16#A3F5, 16#A3F6, 16#A3F7, 16#A3F8, 16#A3F9, 16#A3FA, 16#A3FB, 16#A3FC, 16#A3FD, 16#A1AB, 16#A1E9, 16#A1EA, 16#A3FE, 16#A3A4, 2(0)];
   END_VAR

   VAR_TEMP
      i : UDInt;
      j : UDInt;
      li : UDInt;
      hi : UDInt;
   END_VAR


BEGIN
	IF #UNICODE < 16#0080 THEN
	    #GB2312 := #UNICODE;
	ELSE
	    #hi := 7480;
	    #li := 0;
	    FOR #j := 0 TO 13 BY 1 DO
	        #i := #li + (#hi - #li) / 2;
	        IF #UNICODE = #UNI[#i] THEN
	            #GB2312 := #GB2[#i];
	            EXIT;
	        END_IF;
	        IF #UNICODE > #UNI[#i] THEN
	            #li := #i;
	        ELSE
	            #hi := #i;
	        END_IF;
	    END_FOR;
	END_IF;
END_FUNCTION_BLOCK

FUNCTION_BLOCK "UTF8_TO_GB2312"
{ S7_Optimized_Access := 'TRUE' }
VERSION : 0.1
   VAR_INPUT
      UTF8 : String[254];
   END_VAR

   VAR_OUTPUT
      GB2312 : String[254];
   END_VAR

   VAR
      u8_u { S7_SetPoint := 'False'} : "UTF8_TO_UNI";
      u_g : "UNI_TO_GB2";
   END_VAR

   VAR_TEMP
      i : Int;
      j : Int;
      lenUTF8 : Int;
      tempword : Word;
      tempstr : String[5];
   END_VAR


BEGIN
	#GB2312 := '';
	#tempstr := '0000';
	#lenUTF8 := LEN(#UTF8);
	IF #lenUTF8 > 0 THEN
	    #j := 1;
	    FOR #i := 1 TO #lenUTF8 DO
	        IF #i = #j THEN
	            IF BYTE_TO_WORD(#UTF8[#i]) < 16#0080 THEN
	                #tempstr := MID(IN := #UTF8, L := 1, P := #i);
	                #j := #j + 1;
	            ELSIF BYTE_TO_WORD(#UTF8[#i]) >= 16#C0 AND BYTE_TO_WORD(#UTF8[#i]) < 16#E0 THEN
	                #tempstr := MID(IN := #UTF8, L := 2, P := #i);
	                #j := #j + 2;
	            ELSIF BYTE_TO_WORD(#UTF8[#i]) >= 16#E0 AND BYTE_TO_WORD(#UTF8[#i]) < 16#F0 THEN
	                #tempstr := MID(IN := #UTF8, L := 3, P := #i);
	                #j := #j + 3;
	            ELSIF BYTE_TO_WORD(#UTF8[#i]) >= 16#F0 AND BYTE_TO_WORD(#UTF8[#i]) < 16#F8 THEN
	                #tempstr := MID(IN := #UTF8, L := 4, P := #i);
	                #j := #j + 4;
	            END_IF;
	            IF BYTE_TO_WORD(#UTF8[#i]) >= 16#0080 THEN
	                #u8_u(UTF8 := #tempstr,
	                      UNICODE => #tempword);
	                #u_g(UNICODE := #tempword,
	                     GB2312 => #tempword);
	                #tempstr[2] := WORD_TO_BYTE(#tempword AND 16#FF);
	                #tempstr[1] := WORD_TO_BYTE(SHR(IN := #tempword, N := 8) AND 16#FF);
	                #tempstr := LEFT(IN := #tempstr, L := 2);
	            END_IF;
	            #GB2312 := CONCAT(IN1 := #GB2312, IN2 := #tempstr);
	        END_IF;
	    END_FOR;
	END_IF;
END_FUNCTION_BLOCK

